	W =  90.000 deg,	P =   0.000 deg,	R =   90.000 deg
};
P[1718]{
   GP1:
	UF : 0, UT : 6,		CONFIG : 'N U T, 0, 0, 0',
	X =  65.499  mm,	Y =   -283.961  mm,	Z =   -229.185  mm,
	W =  90.000 deg,	P =   0.000 deg,	R =   90.000 deg
};
P[1719]{
   GP1:
	UF : 0, UT : 6,		CONFIG : 'N U T, 0, 0, 0',
	X =  64.374  mm,	Y =   -284.663  mm,	Z =   -229.314  mm,
	W =  90.000 deg,	P =   0.000 deg,	R =   90.000 deg
};
P[1720]{
   GP1:
	UF : 0, UT : 6,		CONFIG : 'N U T, 0, 0, 0',
	X =  62.334  mm,	Y =   -285.736  mm,	Z =   -229.059  mm,
	W =  90.000 deg,	P =   0.000 deg,	R =   90.000 deg
};
P[1721]{
   GP1:
	UF : 0, UT : 6,		CONFIG : 'N U T, 0, 0, 0',
	X =  61.528  mm,	Y =   -286.336  mm,	Z =   -229.385  mm,
	W =  90.000 deg,	P =   0.000 deg,	R =   90.000 deg
};
P[1722]{
   GP1:
	UF : 0, UT : 6,		CONFIG : 'N U T, 0, 0, 0',
	X =  60.500  mm,	Y =   -286.765  mm,	Z =   -228.984  mm,
	W =  90.000 deg,	P =   0.000 deg,	R =   90.000 deg
};
P[1723]{
   GP1:
	UF : 0, UT : 6,		CONFIG : 'N U T, 0, 0, 0',
	X =  59.972  mm,	Y =   -287.179  mm,	Z =   -229.250  mm,
	W =  90.000 deg,	P =   0.000 deg,	R =   90.000 deg
};
P[1724]{
   GP1:
	UF : 0, UT : 6,		CONFIG : 'N U T, 0, 0, 0',
	X =  58.339  mm,	Y =   -288.171  mm,	Z =   -229.370  mm,
	W =  90.000 deg,	P =   0.000 deg,	R =   90.000 deg
};
P[1725]{
   GP1:
	UF : 0, UT : 6,		CONFIG : 'N U T, 0, 0, 0',
	X =  53.179  mm,	Y =   -291.104  mm,	Z =   -229.258  mm,
	W =  90.000 deg,	P =   0.000 deg,	R =   90.000 deg
};
P[1726]{
   GP1:
	UF : 0, UT : 6,		CONFIG : 'N U T, 0, 0, 0',
	X =  52.446  mm,	Y =   -291.487  mm,	Z =   -229.159  mm,
	W =  90.000 deg,	P =   0.000 deg,	R =   90.000 deg
};
P[1727]{
   GP1:
	UF : 0, UT : 6,		CONFIG : 'N U T, 0, 0, 0',
	X =  50.068  mm,	Y =   -292.765  mm,	Z =   -228.929  mm,
	W =  90.000 deg,	P =   0.000 deg,	R =   90.000 deg
};
P[1728]{
   GP1:
	UF : 0, UT : 6,		CONFIG : 'N U T, 0, 0, 0',
	X =  47.155  mm,	Y =   -294.447  mm,	Z =   -228.929  mm,
	W =  90.000 deg,	P =   0.000 deg,	R =   90.000 deg
};
P[1729]{
   GP1:
	UF : 0, UT : 6,		CONFIG : 'N U T, 0, 0, 0',
	X =  45.389  mm,	Y =   -295.537  mm,	Z =   -229.099  mm,
	W =  90.000 deg,	P =   0.000 deg,	R =   90.000 deg
};
P[1730]{
   GP1:
	UF : 0, UT : 6,		CONFIG : 'N U T, 0, 0, 0',
	X =  41.975  mm,	Y =   -297.626  mm,	Z =   -229.386  mm,
	W =  90.000 deg,	P =   0.000 deg,	R =   90.000 deg
};
P[1731]{
   GP1:
	UF : 0, UT : 6,		CONFIG : 'N U T, 0, 0, 0',
	X =  40.743  mm,	Y =   -298.267  mm,	Z =   -229.217  mm,
	W =  90.000 deg,	P =   0.000 deg,	R =   90.000 deg
};
P[1732]{
   GP1:
	UF : 0, UT : 6,		CONFIG : 'N U T, 0, 0, 0',
	X =  39.529  mm,	Y =   -298.978  mm,	Z =   -229.239  mm,
	W =  90.000 deg,	P =   0.000 deg,	R =   90.000 deg
};
P[1733]{
   GP1:
	UF : 0, UT : 6,		CONFIG : 'N U T, 0, 0, 0',
	X =  38.765  mm,	Y =   -299.424  mm,	Z =   -229.251  mm,
	W =  90.000 deg,	P =   0.000 deg,	R =   90.000 deg
};
P[1734]{
   GP1:
	UF : 0, UT : 6,		CONFIG : 'N U T, 0, 0, 0',
	X =  37.888  mm,	Y =   -299.974  mm,	Z =   -229.356  mm,
	W =  90.000 deg,	P =   0.000 deg,	R =   90.000 deg
};
P[1735]{
   GP1:
	UF : 0, UT : 6,		CONFIG : 'N U T, 0, 0, 0',
	X =  37.310  mm,	Y =   -300.268  mm,	Z =   -229.259  mm,
	W =  90.000 deg,	P =   0.000 deg,	R =   90.000 deg
};
P[1736]{
   GP1:
	UF : 0, UT : 6,		CONFIG : 'N U T, 0, 0, 0',
	X =  36.423  mm,	Y =   -300.815  mm,	Z =   -229.344  mm,
	W =  90.000 deg,	P =   0.000 deg,	R =   90.000 deg
};
P[1737]{
   GP1:
	UF : 0, UT : 6,		CONFIG : 'N U T, 0, 0, 0',
	X =  34.210  mm,	Y =   -301.938  mm,	Z =   -228.969  mm,
	W =  90.000 deg,	P =   0.000 deg,	R =   90.000 deg
};
P[1738]{
   GP1:
	UF : 0, UT : 6,		CONFIG : 'N U T, 0, 0, 0',
	X =  31.437  mm,	Y =   -303.526  mm,	Z =   -228.939  mm,
	W =  90.000 deg,	P =   0.000 deg,	R =   90.000 deg
};
P[1739]{
   GP1:
	UF : 0, UT : 6,		CONFIG : 'N U T, 0, 0, 0',
	X =  30.762  mm,	Y =   -303.936  mm,	Z =   -228.988  mm,
	W =  90.000 deg,	P =   0.000 deg,	R =   90.000 deg
};
P[1740]{
   GP1:
	UF : 0, UT : 6,		CONFIG : 'N U T, 0, 0, 0',
	X =  30.126  mm,	Y =   -304.358  mm,	Z =   -229.121  mm,
	W =  90.000 deg,	P =   0.000 deg,	R =   90.000 deg
};
P[1741]{
   GP1:
	UF : 0, UT : 6,		CONFIG : 'N U T, 0, 0, 0',
	X =  29.321  mm,	Y =   -304.858  mm,	Z =   -229.206  mm,
	W =  90.000 deg,	P =   0.000 deg,	R =   90.000 deg
};
P[1742]{
   GP1:
	UF : 0, UT : 6,		CONFIG : 'N U T, 0, 0, 0',
	X =  28.546  mm,	Y =   -305.311  mm,	Z =   -229.219  mm,
	W =  90.000 deg,	P =   0.000 deg,	R =   90.000 deg
};
P[1743]{
   GP1:
	UF : 0, UT : 6,		CONFIG : 'N U T, 0, 0, 0',
	X =  26.880  mm,	Y =   -306.323  mm,	Z =   -229.338  mm,
	W =  90.000 deg,	P =   0.000 deg,	R =   90.000 deg
};
P[1744]{
   GP1:
	UF : 0, UT : 6,		CONFIG : 'N U T, 0, 0, 0',
	X =  24.918  mm,	Y =   -307.459  mm,	Z =   -229.349  mm,
	W =  90.000 deg,	P =   0.000 deg,	R =   90.000 deg
};
P[1745]{
   GP1:
	UF : 0, UT : 6,		CONFIG : 'N U T, 0, 0, 0',
	X =  24.359  mm,	Y =   -307.779  mm,	Z =   -229.343  mm,
	W =  90.000 deg,	P =   0.000 deg,	R =   90.000 deg
};
P[1746]{
   GP1:
	UF : 0, UT : 6,		CONFIG : 'N U T, 0, 0, 0',
	X =  23.494  mm,	Y =   -308.206  mm,	Z =   -229.165  mm,
	W =  90.000 deg,	P =   0.000 deg,	R =   90.000 deg
};
P[1747]{
   GP1:
	UF : 0, UT : 6,		CONFIG : 'N U T, 0, 0, 0',
	X =  22.302  mm,	Y =   -308.926  mm,	Z =   -229.240  mm,
	W =  90.000 deg,	P =   0.000 deg,	R =   90.000 deg
};
P[1748]{
   GP1:
	UF : 0, UT : 6,		CONFIG : 'N U T, 0, 0, 0',
	X =  20.679  mm,	Y =   -309.863  mm,	Z =   -229.241  mm,
	W =  90.000 deg,	P =   0.000 deg,	R =   90.000 deg
};
P[1749]{
   GP1:
	UF : 0, UT : 6,		CONFIG : 'N U T, 0, 0, 0',
	X =  17.947  mm,	Y =   -311.366  mm,	Z =   -229.061  mm,
	W =  90.000 deg,	P =   0.000 deg,	R =   90.000 deg
};
P[1750]{
   GP1:
	UF : 0, UT : 6,		CONFIG : 'N U T, 0, 0, 0',
	X =  15.569  mm,	Y =   -312.760  mm,	Z =   -229.113  mm,
	W =  90.000 deg,	P =   0.000 deg,	R =   90.000 deg
};
P[1751]{
   GP1:
	UF : 0, UT : 6,		CONFIG : 'N U T, 0, 0, 0',
	X =  12.896  mm,	Y =   -314.404  mm,	Z =   -229.357  mm,
	W =  90.000 deg,	P =   0.000 deg,	R =   90.000 deg
};
P[1752]{
   GP1:
	UF : 0, UT : 6,		CONFIG : 'N U T, 0, 0, 0',
	X =  11.173  mm,	Y =   -315.284  mm,	Z =   -229.077  mm,
	W =  90.000 deg,	P =   0.000 deg,	R =   90.000 deg
};
P[1753]{
   GP1:
	UF : 0, UT : 6,		CONFIG : 'N U T, 0, 0, 0',
	X =  9.686  mm,	Y =   -316.168  mm,	Z =   -229.140  mm,
	W =  90.000 deg,	P =   0.000 deg,	R =   90.000 deg
};
P[1754]{
   GP1:
	UF : 0, UT : 6,		CONFIG : 'N U T, 0, 0, 0',
	X =  8.873  mm,	Y =   -316.625  mm,	Z =   -229.112  mm,
	W =  90.000 deg,	P =   0.000 deg,	R =   90.000 deg
};
P[1755]{
   GP1:
	UF : 0, UT : 6,		CONFIG : 'N U T, 0, 0, 0',
	X =  8.041  mm,	Y =   -317.205  mm,	Z =   -229.351  mm,
	W =  90.000 deg,	P =   0.000 deg,	R =   90.000 deg
};
P[1756]{
   GP1:
	UF : 0, UT : 6,		CONFIG : 'N U T, 0, 0, 0',
	X =  6.642  mm,	Y =   -317.970  mm,	Z =   -229.246  mm,
	W =  90.000 deg,	P =   0.000 deg,	R =   90.000 deg
};
P[1757]{
   GP1:
	UF : 0, UT : 6,		CONFIG : 'N U T, 0, 0, 0',
	X =  5.653  mm,	Y =   -318.591  mm,	Z =   -229.370  mm,
	W =  90.000 deg,	P =   0.000 deg,	R =   90.000 deg
};
P[1758]{
   GP1:
	UF : 0, UT : 6,		CONFIG : 'N U T, 0, 0, 0',
	X =  4.796  mm,	Y =   -318.944  mm,	Z =   -229.023  mm,
	W =  90.000 deg,	P =   0.000 deg,	R =   90.000 deg
};
P[1759]{
   GP1:
	UF : 0, UT : 6,		CONFIG : 'N U T, 0, 0, 0',
	X =  3.388  mm,	Y =   -319.857  mm,	Z =   -229.269  mm,
	W =  90.000 deg,	P =   0.000 deg,	R =   90.000 deg
};
P[1760]{
   GP1:
	UF : 0, UT : 6,		CONFIG : 'N U T, 0, 0, 0',
	X =  2.077  mm,	Y =   -320.526  mm,	Z =   -229.055  mm,
	W =  90.000 deg,	P =   0.000 deg,	R =   90.000 deg
};
P[1761]{
   GP1:
	UF : 0, UT : 6,		CONFIG : 'N U T, 0, 0, 0',
	X =  0.657  mm,	Y =   -321.382  mm,	Z =   -229.142  mm,
	W =  90.000 deg,	P =   0.000 deg,	R =   90.000 deg
};
P[1762]{
   GP1:
	UF : 0, UT : 6,		CONFIG : 'N U T, 0, 0, 0',
	X =  -0.741  mm,	Y =   -322.160  mm,	Z =   -229.070  mm,
	W =  90.000 deg,	P =   0.000 deg,	R =   90.000 deg
};
P[1763]{
   GP1:
	UF : 0, UT : 6,		CONFIG : 'N U T, 0, 0, 0',
	X =  -1.523  mm,	Y =   -322.657  mm,	Z =   -229.181  mm,
	W =  90.000 deg,	P =   0.000 deg,	R =   90.000 deg
};
P[1764]{
   GP1:
	UF : 0, UT : 6,		CONFIG : 'N U T, 0, 0, 0',
	X =  -2.343  mm,	Y =   -323.167  mm,	Z =   -229.270  mm,
	W =  90.000 deg,	P =   0.000 deg,	R =   90.000 deg
};
P[1765]{
   GP1:
	UF : 0, UT : 6,		CONFIG : 'N U T, 0, 0, 0',
	X =  -3.964  mm,	Y =   -323.984  mm,	Z =   -228.981  mm,
	W =  90.000 deg,	P =   0.000 deg,	R =   90.000 deg
};
P[1766]{
   GP1:
	UF : 0, UT : 6,		CONFIG : 'N U T, 0, 0, 0',
	X =  -6.538  mm,	Y =   -325.534  mm,	Z =   -229.136  mm,
	W =  90.000 deg,	P =   0.000 deg,	R =   90.000 deg
};
P[1767]{
   GP1:
	UF : 0, UT : 6,		CONFIG : 'N U T, 0, 0, 0',
	X =  -7.592  mm,	Y =   -326.225  mm,	Z =   -229.338  mm,
	W =  90.000 deg,	P =   0.000 deg,	R =   90.000 deg
};
P[1768]{
   GP1:
	UF : 0, UT : 6,		CONFIG : 'N U T, 0, 0, 0',
	X =  -12.691  mm,	Y =   -329.122  mm,	Z =   -229.220  mm,
	W =  90.000 deg,	P =   0.000 deg,	R =   90.000 deg
};
P[1769]{
   GP1:
	UF : 0, UT : 6,		CONFIG : 'N U T, 0, 0, 0',
	X =  -13.895  mm,	Y =   -329.816  mm,	Z =   -229.218  mm,
	W =  90.000 deg,	P =   0.000 deg,	R =   90.000 deg
};
P[1770]{
   GP1:
	UF : 0, UT : 6,		CONFIG : 'N U T, 0, 0, 0',
	X =  -14.816  mm,	Y =   -330.402  mm,	Z =   -229.349  mm,
	W =  90.000 deg,	P =   0.000 deg,	R =   90.000 deg
};
P[1771]{
   GP1:
	UF : 0, UT : 6,		CONFIG : 'N U T, 0, 0, 0',
	X =  -15.958  mm,	Y =   -330.974  mm,	Z =   -229.139  mm,
	W =  90.000 deg,	P =   0.000 deg,	R =   90.000 deg
};
P[1772]{
   GP1:
	UF : 0, UT : 6,		CONFIG : 'N U T, 0, 0, 0',
	X =  -17.640  mm,	Y =   -331.967  mm,	Z =   -229.191  mm,
	W =  90.000 deg,	P =   0.000 deg,	R =   90.000 deg
};
P[1773]{
   GP1:
	UF : 0, UT : 6,		CONFIG : 'N U T, 0, 0, 0',
	X =  -19.082  mm,	Y =   -332.836  mm,	Z =   -229.281  mm,
	W =  90.000 deg,	P =   0.000 deg,	R =   90.000 deg
};
P[1774]{
   GP1:
	UF : 0, UT : 6,		CONFIG : 'N U T, 0, 0, 0',
	X =  -19.863  mm,	Y =   -333.279  mm,	Z =   -229.261  mm,
	W =  90.000 deg,	P =   0.000 deg,	R =   90.000 deg
};
P[1775]{
   GP1:
	UF : 0, UT : 6,		CONFIG : 'N U T, 0, 0, 0',
	X =  -21.186  mm,	Y =   -333.972  mm,	Z =   -229.088  mm,
	W =  90.000 deg,	P =   0.000 deg,	R =   90.000 deg
};
P[1776]{
   GP1:
	UF : 0, UT : 6,		CONFIG : 'N U T, 0, 0, 0',
	X =  -22.635  mm,	Y =   -334.894  mm,	Z =   -229.296  mm,
	W =  90.000 deg,	P =   0.000 deg,	R =   90.000 deg
};
P[1777]{
   GP1:
	UF : 0, UT : 6,		CONFIG : 'N U T, 0, 0, 0',
	X =  -24.157  mm,	Y =   -335.703  mm,	Z =   -229.127  mm,
	W =  90.000 deg,	P =   0.000 deg,	R =   90.000 deg
};
P[1778]{
   GP1:
	UF : 0, UT : 6,		CONFIG : 'N U T, 0, 0, 0',
	X =  -25.039  mm,	Y =   -336.224  mm,	Z =   -229.155  mm,
	W =  90.000 deg,	P =   0.000 deg,	R =   90.000 deg
};
P[1779]{
   GP1:
	UF : 0, UT : 6,		CONFIG : 'N U T, 0, 0, 0',
	X =  -25.704  mm,	Y =   -336.510  mm,	Z =   -228.916  mm,
	W =  90.000 deg,	P =   0.000 deg,	R =   90.000 deg
};
P[1780]{
   GP1:
	UF : 0, UT : 6,		CONFIG : 'N U T, 0, 0, 0',
	X =  -26.496  mm,	Y =   -337.068  mm,	Z =   -229.160  mm,
	W =  90.000 deg,	P =   0.000 deg,	R =   90.000 deg
};
P[1781]{
   GP1:
	UF : 0, UT : 6,		CONFIG : 'N U T, 0, 0, 0',
	X =  -29.082  mm,	Y =   -338.564  mm,	Z =   -229.168  mm,
	W =  90.000 deg,	P =   0.000 deg,	R =   90.000 deg
};
P[1782]{
   GP1:
	UF : 0, UT : 6,		CONFIG : 'N U T, 0, 0, 0',
	X =  -32.694  mm,	Y =   -340.689  mm,	Z =   -229.266  mm,
	W =  90.000 deg,	P =   0.000 deg,	R =   90.000 deg
};
P[1783]{
   GP1:
	UF : 0, UT : 6,		CONFIG : 'N U T, 0, 0, 0',
	X =  -33.349  mm,	Y =   -341.119  mm,	Z =   -229.387  mm,
	W =  90.000 deg,	P =   0.000 deg,	R =   90.000 deg
};
P[1784]{
   GP1:
	UF : 0, UT : 6,		CONFIG : 'N U T, 0, 0, 0',
	X =  -38.216  mm,	Y =   -343.745  mm,	Z =   -228.944  mm,
	W =  90.000 deg,	P =   0.000 deg,	R =   90.000 deg
};
P[1785]{
   GP1:
	UF : 0, UT : 6,		CONFIG : 'N U T, 0, 0, 0',
	X =  -41.561  mm,	Y =   -345.684  mm,	Z =   -228.963  mm,
	W =  90.000 deg,	P =   0.000 deg,	R =   90.000 deg
};
P[1786]{
   GP1:
	UF : 0, UT : 6,		CONFIG : 'N U T, 0, 0, 0',
	X =  -42.055  mm,	Y =   -346.140  mm,	Z =   -229.376  mm,
	W =  90.000 deg,	P =   0.000 deg,	R =   90.000 deg
};
P[1787]{
   GP1:
	UF : 0, UT : 6,		CONFIG : 'N U T, 0, 0, 0',
	X =  -42.732  mm,	Y =   -346.389  mm,	Z =   -229.030  mm,
	W =  90.000 deg,	P =   0.000 deg,	R =   90.000 deg
};
P[1788]{
   GP1:
	UF : 0, UT : 6,		CONFIG : 'N U T, 0, 0, 0',
	X =  -43.777  mm,	Y =   -347.079  mm,	Z =   -229.241  mm,
	W =  90.000 deg,	P =   0.000 deg,	R =   90.000 deg
};
P[1789]{
   GP1:
	UF : 0, UT : 6,		CONFIG : 'N U T, 0, 0, 0',
	X =  -44.518  mm,	Y =   -347.535  mm,	Z =   -229.311  mm,
	W =  90.000 deg,	P =   0.000 deg,	R =   90.000 deg
};
P[1790]{
   GP1:
	UF : 0, UT : 6,		CONFIG : 'N U T, 0, 0, 0',
	X =  -45.258  mm,	Y =   -347.966  mm,	Z =   -229.318  mm,
	W =  90.000 deg,	P =   0.000 deg,	R =   90.000 deg
};
P[1791]{
   GP1:
	UF : 0, UT : 6,		CONFIG : 'N U T, 0, 0, 0',
	X =  -46.748  mm,	Y =   -348.709  mm,	Z =   -229.034  mm,
	W =  90.000 deg,	P =   0.000 deg,	R =   90.000 deg
};
P[1792]{
   GP1:
	UF : 0, UT : 6,		CONFIG : 'N U T, 0, 0, 0',
	X =  -50.185  mm,	Y =   -350.794  mm,	Z =   -229.276  mm,
	W =  90.000 deg,	P =   0.000 deg,	R =   90.000 deg
};
P[1793]{
   GP1:
	UF : 0, UT : 6,		CONFIG : 'N U T, 0, 0, 0',
	X =  -50.896  mm,	Y =   -351.228  mm,	Z =   -229.333  mm,
	W =  90.000 deg,	P =   0.000 deg,	R =   90.000 deg
};
P[1794]{
   GP1:
	UF : 0, UT : 6,		CONFIG : 'N U T, 0, 0, 0',
	X =  -51.979  mm,	Y =   -351.709  mm,	Z =   -228.984  mm,
	W =  90.000 deg,	P =   0.000 deg,	R =   90.000 deg
};
P[1795]{
   GP1:
	UF : 0, UT : 6,		CONFIG : 'N U T, 0, 0, 0',
	X =  -54.128  mm,	Y =   -353.013  mm,	Z =   -229.137  mm,
	W =  90.000 deg,	P =   0.000 deg,	R =   90.000 deg
};
P[1796]{
   GP1:
	UF : 0, UT : 6,		CONFIG : 'N U T, 0, 0, 0',
	X =  -54.799  mm,	Y =   -353.441  mm,	Z =   -229.237  mm,
	W =  90.000 deg,	P =   0.000 deg,	R =   90.000 deg
};
P[1797]{
   GP1:
	UF : 0, UT : 6,		CONFIG : 'N U T, 0, 0, 0',
	X =  -55.346  mm,	Y =   -353.813  mm,	Z =   -229.371  mm,
	W =  90.000 deg,	P =   0.000 deg,	R =   90.000 deg
};
P[1798]{
   GP1:
	UF : 0, UT : 6,		CONFIG : 'N U T, 0, 0, 0',
	X =  -59.610  mm,	Y =   -356.160  mm,	Z =   -229.092  mm,
	W =  90.000 deg,	P =   0.000 deg,	R =   90.000 deg
};
P[1799]{
   GP1:
	UF : 0, UT : 6,		CONFIG : 'N U T, 0, 0, 0',
	X =  -60.201  mm,	Y =   -356.446  mm,	Z =   -228.959  mm,
	W =  90.000 deg,	P =   0.000 deg,	R =   90.000 deg
};
P[1800]{
   GP1:
	UF : 0, UT : 6,		CONFIG : 'N U T, 0, 0, 0',
	X =  -61.122  mm,	Y =   -357.104  mm,	Z =   -229.266  mm,
	W =  90.000 deg,	P =   0.000 deg,	R =   90.000 deg
};
P[1801]{
   GP1:
	UF : 0, UT : 6,		CONFIG : 'N U T, 0, 0, 0',
	X =  -62.393  mm,	Y =   -357.747  mm,	Z =   -229.045  mm,
	W =  90.000 deg,	P =   0.000 deg,	R =   90.000 deg
};
P[1802]{
   GP1:
	UF : 0, UT : 6,		CONFIG : 'N U T, 0, 0, 0',
	X =  -63.618  mm,	Y =   -358.533  mm,	Z =   -229.238  mm,
	W =  90.000 deg,	P =   0.000 deg,	R =   90.000 deg
};
P[1803]{
   GP1:
	UF : 0, UT : 6,		CONFIG : 'N U T, 0, 0, 0',
	X =  -64.685  mm,	Y =   -359.172  mm,	Z =   -229.293  mm,
	W =  90.000 deg,	P =   0.000 deg,	R =   90.000 deg
};
P[1804]{
   GP1:
	UF : 0, UT : 6,		CONFIG : 'N U T, 0, 0, 0',
	X =  -65.434  mm,	Y =   -359.590  mm,	Z =   -229.257  mm,
	W =  90.000 deg,	P =   0.000 deg,	R =   90.000 deg
};
P[1805]{
   GP1:
	UF : 0, UT : 6,		CONFIG : 'N U T, 0, 0, 0',
	X =  -67.552  mm,	Y =   -360.821  mm,	Z =   -229.277  mm,
	W =  90.000 deg,	P =   0.000 deg,	R =   90.000 deg
};
P[1806]{
   GP1:
	UF : 0, UT : 6,		CONFIG : 'N U T, 0, 0, 0',
	X =  -68.252  mm,	Y =   -361.161  mm,	Z =   -229.121  mm,
	W =  90.000 deg,	P =   0.000 deg,	R =   90.000 deg
};
P[1807]{
   GP1:
	UF : 0, UT : 6,		CONFIG : 'N U T, 0, 0, 0',
	X =  -69.737  mm,	Y =   -361.996  mm,	Z =   -229.066  mm,
	W =  90.000 deg,	P =   0.000 deg,	R =   90.000 deg
};
P[1808]{
   GP1:
	UF : 0, UT : 6,		CONFIG : 'N U T, 0, 0, 0',
	X =  -71.695  mm,	Y =   -363.184  mm,	Z =   -229.206  mm,
	W =  90.000 deg,	P =   0.000 deg,	R =   90.000 deg
};
P[1809]{
   GP1:
	UF : 0, UT : 6,		CONFIG : 'N U T, 0, 0, 0',
	X =  -73.384  mm,	Y =   -364.195  mm,	Z =   -229.294  mm,
	W =  90.000 deg,	P =   0.000 deg,	R =   90.000 deg
};
P[1810]{
   GP1:
	UF : 0, UT : 6,		CONFIG : 'N U T, 0, 0, 0',
	X =  -74.673  mm,	Y =   -364.878  mm,	Z =   -229.144  mm,
	W =  90.000 deg,	P =   0.000 deg,	R =   90.000 deg
};
P[1811]{
   GP1:
	UF : 0, UT : 6,		CONFIG : 'N U T, 0, 0, 0',
	X =  -76.471  mm,	Y =   -365.928  mm,	Z =   -229.173  mm,
	W =  90.000 deg,	P =   0.000 deg,	R =   90.000 deg
};
P[1812]{
   GP1:
	UF : 0, UT : 6,		CONFIG : 'N U T, 0, 0, 0',
	X =  -78.015  mm,	Y =   -366.782  mm,	Z =   -229.082  mm,
	W =  90.000 deg,	P =   0.000 deg,	R =   90.000 deg
};
P[1813]{
   GP1:
	UF : 0, UT : 6,		CONFIG : 'N U T, 0, 0, 0',
	X =  -82.837  mm,	Y =   -369.534  mm,	Z =   -229.004  mm,
	W =  90.000 deg,	P =   0.000 deg,	R =   90.000 deg
};
P[1814]{
   GP1:
	UF : 0, UT : 6,		CONFIG : 'N U T, 0, 0, 0',
	X =  -83.583  mm,	Y =   -369.935  mm,	Z =   -228.932  mm,
	W =  90.000 deg,	P =   0.000 deg,	R =   90.000 deg
};
P[1815]{
   GP1:
	UF : 0, UT : 6,		CONFIG : 'N U T, 0, 0, 0',
	X =  -85.190  mm,	Y =   -370.941  mm,	Z =   -229.121  mm,
	W =  90.000 deg,	P =   0.000 deg,	R =   90.000 deg
};
P[1816]{
   GP1:
	UF : 0, UT : 6,		CONFIG : 'N U T, 0, 0, 0',
	X =  -86.946  mm,	Y =   -371.886  mm,	Z =   -228.955  mm,
	W =  90.000 deg,	P =   0.000 deg,	R =   90.000 deg
};
P[1817]{
   GP1:
	UF : 0, UT : 6,		CONFIG : 'N U T, 0, 0, 0',
	X =  -87.736  mm,	Y =   -372.509  mm,	Z =   -229.360  mm,
	W =  90.000 deg,	P =   0.000 deg,	R =   90.000 deg
};
P[1818]{
   GP1:
	UF : 0, UT : 6,		CONFIG : 'N U T, 0, 0, 0',
	X =  -89.887  mm,	Y =   -373.748  mm,	Z =   -229.351  mm,
	W =  90.000 deg,	P =   0.000 deg,	R =   90.000 deg
};
P[1819]{
   GP1:
	UF : 0, UT : 6,		CONFIG : 'N U T, 0, 0, 0',
	X =  -91.030  mm,	Y =   -374.267  mm,	Z =   -229.010  mm,
	W =  90.000 deg,	P =   0.000 deg,	R =   90.000 deg
};
P[1820]{
   GP1:
	UF : 0, UT : 6,		CONFIG : 'N U T, 0, 0, 0',
	X =  -94.361  mm,	Y =   -376.300  mm,	Z =   -229.274  mm,
	W =  90.000 deg,	P =   0.000 deg,	R =   90.000 deg
};
P[1821]{
   GP1:
	UF : 0, UT : 6,		CONFIG : 'N U T, 0, 0, 0',
	X =  -96.414  mm,	Y =   -377.422  mm,	Z =   -229.121  mm,
	W =  90.000 deg,	P =   0.000 deg,	R =   90.000 deg
};
P[1822]{
   GP1:
	UF : 0, UT : 6,		CONFIG : 'N U T, 0, 0, 0',
	X =  -98.002  mm,	Y =   -378.340  mm,	Z =   -229.123  mm,
	W =  90.000 deg,	P =   0.000 deg,	R =   90.000 deg
};
P[1823]{
   GP1:
	UF : 0, UT : 6,		CONFIG : 'N U T, 0, 0, 0',
	X =  -101.725  mm,	Y =   -380.543  mm,	Z =   -229.255  mm,
	W =  90.000 deg,	P =   0.000 deg,	R =   90.000 deg
};
P[1824]{
   GP1:
	UF : 0, UT : 6,		CONFIG : 'N U T, 0, 0, 0',
	X =  -102.580  mm,	Y =   -381.019  mm,	Z =   -229.211  mm,
	W =  90.000 deg,	P =   0.000 deg,	R =   90.000 deg
};
P[1825]{
   GP1:
	UF : 0, UT : 6,		CONFIG : 'N U T, 0, 0, 0',
	X =  -103.214  mm,	Y =   -381.274  mm,	Z =   -228.942  mm,
	W =  90.000 deg,	P =   0.000 deg,	R =   90.000 deg
};
P[1826]{
   GP1:
	UF : 0, UT : 6,		CONFIG : 'N U T, 0, 0, 0',
	X =  -104.057  mm,	Y =   -381.765  mm,	Z =   -228.951  mm,
	W =  90.000 deg,	P =   0.000 deg,	R =   90.000 deg
};
P[1827]{
   GP1:
	UF : 0, UT : 6,		CONFIG : 'N U T, 0, 0, 0',
	X =  -104.771  mm,	Y =   -382.207  mm,	Z =   -229.023  mm,
	W =  90.000 deg,	P =   0.000 deg,	R =   90.000 deg
};
P[1828]{
   GP1:
	UF : 0, UT : 6,		CONFIG : 'N U T, 0, 0, 0',
	X =  -106.220  mm,	Y =   -383.159  mm,	Z =   -229.305  mm,
	W =  90.000 deg,	P =   0.000 deg,	R =   90.000 deg
};
P[1829]{
   GP1:
	UF : 0, UT : 6,		CONFIG : 'N U T, 0, 0, 0',
	X =  -107.258  mm,	Y =   -383.655  mm,	Z =   -229.053  mm,
	W =  90.000 deg,	P =   0.000 deg,	R =   90.000 deg
};
P[1830]{
   GP1:
	UF : 0, UT : 6,		CONFIG : 'N U T, 0, 0, 0',
	X =  -108.626  mm,	Y =   -384.389  mm,	Z =   -228.918  mm,
	W =  90.000 deg,	P =   0.000 deg,	R =   90.000 deg
};
P[1831]{
   GP1:
	UF : 0, UT : 6,		CONFIG : 'N U T, 0, 0, 0',
	X =  -110.424  mm,	Y =   -385.480  mm,	Z =   -229.046  mm,
	W =  90.000 deg,	P =   0.000 deg,	R =   90.000 deg
};
P[1832]{
   GP1:
	UF : 0, UT : 6,		CONFIG : 'N U T, 0, 0, 0',
	X =  -111.106  mm,	Y =   -385.858  mm,	Z =   -228.907  mm,
	W =  90.000 deg,	P =   0.000 deg,	R =   90.000 deg
};
P[1833]{
   GP1:
	UF : 0, UT : 6,		CONFIG : 'N U T, 0, 0, 0',
	X =  -111.846  mm,	Y =   -386.429  mm,	Z =   -229.006  mm,
	W =  90.000 deg,	P =   0.000 deg,	R =   90.000 deg
};
P[1834]{
   GP1:
	UF : 0, UT : 6,		CONFIG : 'N U T, 0, 0, 0',
	X =  -114.050  mm,	Y =   -388.372  mm,	Z =   -229.002  mm,
	W =  90.000 deg,	P =   0.000 deg,	R =   90.000 deg
};
P[1835]{
   GP1:
	UF : 0, UT : 6,		CONFIG : 'N U T, 0, 0, 0',
	X =  -115.101  mm,	Y =   -389.696  mm,	Z =   -228.999  mm,
	W =  90.000 deg,	P =   0.000 deg,	R =   90.000 deg
};
P[1836]{
   GP1:
	UF : 0, UT : 6,		CONFIG : 'N U T, 0, 0, 0',
	X =  -115.762  mm,	Y =   -390.707  mm,	Z =   -228.966  mm,
	W =  90.000 deg,	P =   0.000 deg,	R =   90.000 deg
};
P[1837]{
   GP1:
	UF : 0, UT : 6,		CONFIG : 'N U T, 0, 0, 0',
	X =  -116.815  mm,	Y =   -393.661  mm,	Z =   -229.189  mm,
	W =  90.000 deg,	P =   0.000 deg,	R =   90.000 deg
};
P[1838]{
   GP1:
	UF : 0, UT : 6,		CONFIG : 'N U T, 0, 0, 0',
	X =  -116.981  mm,	Y =   -394.369  mm,	Z =   -229.133  mm,
	W =  90.000 deg,	P =   0.000 deg,	R =   90.000 deg
};
P[1839]{
   GP1:
	UF : 0, UT : 6,		CONFIG : 'N U T, 0, 0, 0',
	X =  -117.216  mm,	Y =   -397.476  mm,	Z =   -229.036  mm,
	W =  90.000 deg,	P =   0.000 deg,	R =   90.000 deg
};
P[1840]{
   GP1:
	UF : 0, UT : 6,		CONFIG : 'N U T, 0, 0, 0',
	X =  -117.144  mm,	Y =   -398.247  mm,	Z =   -229.117  mm,
	W =  90.000 deg,	P =   0.000 deg,	R =   90.000 deg
};
P[1841]{
   GP1:
	UF : 0, UT : 6,		CONFIG : 'N U T, 0, 0, 0',
	X =  -116.699  mm,	Y =   -400.629  mm,	Z =   -228.902  mm,
	W =  90.000 deg,	P =   0.000 deg,	R =   90.000 deg
};
P[1842]{
   GP1:
	UF : 0, UT : 6,		CONFIG : 'N U T, 0, 0, 0',
	X =  -115.143  mm,	Y =   -403.741  mm,	Z =   -229.218  mm,
	W =  90.000 deg,	P =   0.000 deg,	R =   90.000 deg
};
P[1843]{
   GP1:
	UF : 0, UT : 6,		CONFIG : 'N U T, 0, 0, 0',
	X =  -114.830  mm,	Y =   -404.473  mm,	Z =   -228.955  mm,
	W =  90.000 deg,	P =   0.000 deg,	R =   90.000 deg
};
P[1844]{
   GP1:
	UF : 0, UT : 6,		CONFIG : 'N U T, 0, 0, 0',
	X =  -114.278  mm,	Y =   -405.145  mm,	Z =   -229.351  mm,
	W =  90.000 deg,	P =   0.000 deg,	R =   90.000 deg
};
P[1845]{
   GP1:
	UF : 0, UT : 6,		CONFIG : 'N U T, 0, 0, 0',
	X =  -113.583  mm,	Y =   -406.477  mm,	Z =   -229.173  mm,
	W =  90.000 deg,	P =   0.000 deg,	R =   90.000 deg
};
P[1846]{
   GP1:
	UF : 0, UT : 6,		CONFIG : 'N U T, 0, 0, 0',
	X =  -111.947  mm,	Y =   -409.195  mm,	Z =   -229.335  mm,
	W =  90.000 deg,	P =   0.000 deg,	R =   90.000 deg
};
P[1847]{
   GP1:
	UF : 0, UT : 6,		CONFIG : 'N U T, 0, 0, 0',
	X =  -110.907  mm,	Y =   -411.061  mm,	Z =   -229.245  mm,
	W =  90.000 deg,	P =   0.000 deg,	R =   90.000 deg
};
P[1848]{
   GP1:
	UF : 0, UT : 6,		CONFIG : 'N U T, 0, 0, 0',
	X =  -110.205  mm,	Y =   -412.176  mm,	Z =   -229.385  mm,
	W =  90.000 deg,	P =   0.000 deg,	R =   90.000 deg
};
P[1849]{
   GP1:
	UF : 0, UT : 6,		CONFIG : 'N U T, 0, 0, 0',
	X =  -109.969  mm,	Y =   -412.840  mm,	Z =   -229.026  mm,
	W =  90.000 deg,	P =   0.000 deg,	R =   90.000 deg
};
P[1850]{
   GP1:
	UF : 0, UT : 6,		CONFIG : 'N U T, 0, 0, 0',
	X =  -108.686  mm,	Y =   -415.006  mm,	Z =   -229.104  mm,
	W =  90.000 deg,	P =   0.000 deg,	R =   90.000 deg
};
P[1851]{
   GP1:
	UF : 0, UT : 6,		CONFIG : 'N U T, 0, 0, 0',
	X =  -108.139  mm,	Y =   -415.790  mm,	Z =   -229.334  mm,
	W =  90.000 deg,	P =   0.000 deg,	R =   90.000 deg
};
P[1852]{
   GP1:
	UF : 0, UT : 6,		CONFIG : 'N U T, 0, 0, 0',
	X =  -107.446  mm,	Y =   -417.150  mm,	Z =   -229.110  mm,
	W =  90.000 deg,	P =   0.000 deg,	R =   90.000 deg
};
P[1853]{
   GP1:
	UF : 0, UT : 6,		CONFIG : 'N U T, 0, 0, 0',
	X =  -106.777  mm,	Y =   -418.198  mm,	Z =   -229.266  mm,
	W =  90.000 deg,	P =   0.000 deg,	R =   90.000 deg
};
P[1854]{
   GP1:
	UF : 0, UT : 6,		CONFIG : 'N U T, 0, 0, 0',
	X =  -105.715  mm,	Y =   -419.969  mm,	Z =   -229.362  mm,
	W =  90.000 deg,	P =   0.000 deg,	R =   90.000 deg
};
P[1855]{
   GP1:
	UF : 0, UT : 6,		CONFIG : 'N U T, 0, 0, 0',
	X =  -102.894  mm,	Y =   -424.877  mm,	Z =   -229.333  mm,
	W =  90.000 deg,	P =   0.000 deg,	R =   90.000 deg
};
P[1856]{
   GP1:
	UF : 0, UT : 6,		CONFIG : 'N U T, 0, 0, 0',
	X =  -101.587  mm,	Y =   -427.111  mm,	Z =   -229.370  mm,
	W =  90.000 deg,	P =   0.000 deg,	R =   90.000 deg
};
P[1857]{
   GP1:
	UF : 0, UT : 6,		CONFIG : 'N U T, 0, 0, 0',
	X =  -101.111  mm,	Y =   -428.222  mm,	Z =   -228.971  mm,
	W =  90.000 deg,	P =   0.000 deg,	R =   90.000 deg
};
P[1858]{
   GP1:
	UF : 0, UT : 6,		CONFIG : 'N U T, 0, 0, 0',
	X =  -100.738  mm,	Y =   -428.828  mm,	Z =   -229.025  mm,
	W =  90.000 deg,	P =   0.000 deg,	R =   90.000 deg
};
P[1859]{
   GP1:
	UF : 0, UT : 6,		CONFIG : 'N U T, 0, 0, 0',
	X =  -100.382  mm,	Y =   -429.496  mm,	Z =   -228.954  mm,
	W =  90.000 deg,	P =   0.000 deg,	R =   90.000 deg
};
P[1860]{
   GP1:
	UF : 0, UT : 6,		CONFIG : 'N U T, 0, 0, 0',
	X =  -99.771  mm,	Y =   -430.443  mm,	Z =   -229.108  mm,
	W =  90.000 deg,	P =   0.000 deg,	R =   90.000 deg
};
P[1861]{
   GP1:
	UF : 0, UT : 6,		CONFIG : 'N U T, 0, 0, 0',
	X =  -97.945  mm,	Y =   -433.610  mm,	Z =   -229.104  mm,
	W =  90.000 deg,	P =   0.000 deg,	R =   90.000 deg
};
P[1862]{
   GP1:
	UF : 0, UT : 6,		CONFIG : 'N U T, 0, 0, 0',
	X =  -96.878  mm,	Y =   -435.314  mm,	Z =   -229.304  mm,
	W =  90.000 deg,	P =   0.000 deg,	R =   90.000 deg
};
P[1863]{
   GP1:
	UF : 0, UT : 6,		CONFIG : 'N U T, 0, 0, 0',
	X =  -95.918  mm,	Y =   -437.015  mm,	Z =   -229.252  mm,
	W =  90.000 deg,	P =   0.000 deg,	R =   90.000 deg
};
P[1864]{
   GP1:
	UF : 0, UT : 6,		CONFIG : 'N U T, 0, 0, 0',
	X =  -95.734  mm,	Y =   -437.573  mm,	Z =   -228.916  mm,
	W =  90.000 deg,	P =   0.000 deg,	R =   90.000 deg
};
P[1865]{
   GP1:
	UF : 0, UT : 6,		CONFIG : 'N U T, 0, 0, 0',
	X =  -94.251  mm,	Y =   -440.013  mm,	Z =   -229.096  mm,
	W =  90.000 deg,	P =   0.000 deg,	R =   90.000 deg
};
P[1866]{
   GP1:
	UF : 0, UT : 6,		CONFIG : 'N U T, 0, 0, 0',
	X =  -93.487  mm,	Y =   -441.177  mm,	Z =   -229.317  mm,
	W =  90.000 deg,	P =   0.000 deg,	R =   90.000 deg
};
P[1867]{
   GP1:
	UF : 0, UT : 6,		CONFIG : 'N U T, 0, 0, 0',
	X =  -92.630  mm,	Y =   -442.709  mm,	Z =   -229.251  mm,
	W =  90.000 deg,	P =   0.000 deg,	R =   90.000 deg
};
P[1868]{
   GP1:
	UF : 0, UT : 6,		CONFIG : 'N U T, 0, 0, 0',
	X =  -92.385  mm,	Y =   -443.308  mm,	Z =   -229.007  mm,
	W =  90.000 deg,	P =   0.000 deg,	R =   90.000 deg
};
P[1869]{
   GP1:
	UF : 0, UT : 6,		CONFIG : 'N U T, 0, 0, 0',
	X =  -91.614  mm,	Y =   -444.506  mm,	Z =   -229.201  mm,
	W =  90.000 deg,	P =   0.000 deg,	R =   90.000 deg
};
P[1870]{
   GP1:
	UF : 0, UT : 6,		CONFIG : 'N U T, 0, 0, 0',
	X =  -91.022  mm,	Y =   -445.447  mm,	Z =   -229.318  mm,
	W =  90.000 deg,	P =   0.000 deg,	R =   90.000 deg
};
P[1871]{
   GP1:
	UF : 0, UT : 6,		CONFIG : 'N U T, 0, 0, 0',
	X =  -90.796  mm,	Y =   -446.031  mm,	Z =   -229.048  mm,
	W =  90.000 deg,	P =   0.000 deg,	R =   90.000 deg
};
P[1872]{
   GP1:
	UF : 0, UT : 6,		CONFIG : 'N U T, 0, 0, 0',
	X =  -89.661  mm,	Y =   -447.816  mm,	Z =   -229.302  mm,
	W =  90.000 deg,	P =   0.000 deg,	R =   90.000 deg
};
P[1873]{
   GP1:
	UF : 0, UT : 6,		CONFIG : 'N U T, 0, 0, 0',
	X =  -88.469  mm,	Y =   -450.093  mm,	Z =   -229.002  mm,
	W =  90.000 deg,	P =   0.000 deg,	R =   90.000 deg
};
P[1874]{
   GP1:
	UF : 0, UT : 6,		CONFIG : 'N U T, 0, 0, 0',
	X =  -87.738  mm,	Y =   -451.149  mm,	Z =   -229.299  mm,
	W =  90.000 deg,	P =   0.000 deg,	R =   90.000 deg
};
P[1875]{
   GP1:
	UF : 0, UT : 6,		CONFIG : 'N U T, 0, 0, 0',
	X =  -86.732  mm,	Y =   -452.944  mm,	Z =   -229.224  mm,
	W =  90.000 deg,	P =   0.000 deg,	R =   90.000 deg
};
P[1876]{
   GP1:
	UF : 0, UT : 6,		CONFIG : 'N U T, 0, 0, 0',
	X =  -85.455  mm,	Y =   -455.178  mm,	Z =   -229.193  mm,
	W =  90.000 deg,	P =   0.000 deg,	R =   90.000 deg
};
P[1877]{
   GP1:
	UF : 0, UT : 6,		CONFIG : 'N U T, 0, 0, 0',
	X =  -84.898  mm,	Y =   -456.153  mm,	Z =   -229.176  mm,
	W =  90.000 deg,	P =   0.000 deg,	R =   90.000 deg
};
P[1878]{
   GP1:
	UF : 0, UT : 6,		CONFIG : 'N U T, 0, 0, 0',
	X =  -83.663  mm,	Y =   -458.430  mm,	Z =   -228.986  mm,
	W =  90.000 deg,	P =   0.000 deg,	R =   90.000 deg
};
P[1879]{
   GP1:
	UF : 0, UT : 6,		CONFIG : 'N U T, 0, 0, 0',
	X =  -82.928  mm,	Y =   -459.679  mm,	Z =   -229.020  mm,
	W =  90.000 deg,	P =   0.000 deg,	R =   90.000 deg
};
P[1880]{
   GP1:
	UF : 0, UT : 6,		CONFIG : 'N U T, 0, 0, 0',
	X =  -81.085  mm,	Y =   -462.911  mm,	Z =   -228.962  mm,
	W =  90.000 deg,	P =   0.000 deg,	R =   90.000 deg
};
P[1881]{
   GP1:
	UF : 0, UT : 6,		CONFIG : 'N U T, 0, 0, 0',
	X =  -80.232  mm,	Y =   -464.268  mm,	Z =   -229.131  mm,
	W =  90.000 deg,	P =   0.000 deg,	R =   90.000 deg
};
P[1882]{
   GP1:
	UF : 0, UT : 6,		CONFIG : 'N U T, 0, 0, 0',
	X =  -79.260  mm,	Y =   -465.944  mm,	Z =   -229.142  mm,
	W =  90.000 deg,	P =   0.000 deg,	R =   90.000 deg
};
P[1883]{
   GP1:
	UF : 0, UT : 6,		CONFIG : 'N U T, 0, 0, 0',
	X =  -78.133  mm,	Y =   -467.770  mm,	Z =   -229.317  mm,
	W =  90.000 deg,	P =   0.000 deg,	R =   90.000 deg
};
P[1884]{
   GP1:
	UF : 0, UT : 6,		CONFIG : 'N U T, 0, 0, 0',
	X =  -76.870  mm,	Y =   -470.008  mm,	Z =   -229.247  mm,
	W =  90.000 deg,	P =   0.000 deg,	R =   90.000 deg
};
P[1885]{
   GP1:
	UF : 0, UT : 6,		CONFIG : 'N U T, 0, 0, 0',
	X =  -76.601  mm,	Y =   -470.711  mm,	Z =   -228.915  mm,
	W =  90.000 deg,	P =   0.000 deg,	R =   90.000 deg
};
P[1886]{
   GP1:
	UF : 0, UT : 6,		CONFIG : 'N U T, 0, 0, 0',
	X =  -76.006  mm,	Y =   -471.663  mm,	Z =   -229.025  mm,
	W =  90.000 deg,	P =   0.000 deg,	R =   90.000 deg
};
P[1887]{
   GP1:
	UF : 0, UT : 6,		CONFIG : 'N U T, 0, 0, 0',
	X =  -75.413  mm,	Y =   -472.457  mm,	Z =   -229.353  mm,
	W =  90.000 deg,	P =   0.000 deg,	R =   90.000 deg
};
P[1888]{
   GP1:
	UF : 0, UT : 6,		CONFIG : 'N U T, 0, 0, 0',
	X =  -73.867  mm,	Y =   -475.295  mm,	Z =   -229.125  mm,
	W =  90.000 deg,	P =   0.000 deg,	R =   90.000 deg
};
P[1889]{
   GP1:
	UF : 0, UT : 6,		CONFIG : 'N U T, 0, 0, 0',
	X =  -73.257  mm,	Y =   -476.368  mm,	Z =   -229.103  mm,
	W =  90.000 deg,	P =   0.000 deg,	R =   90.000 deg
};
P[1890]{
   GP1:
	UF : 0, UT : 6,		CONFIG : 'N U T, 0, 0, 0',
	X =  -72.393  mm,	Y =   -477.925  mm,	Z =   -229.019  mm,
	W =  90.000 deg,	P =   0.000 deg,	R =   90.000 deg
};
P[1891]{
   GP1:
	UF : 0, UT : 6,		CONFIG : 'N U T, 0, 0, 0',
	X =  -70.648  mm,	Y =   -480.890  mm,	Z =   -229.099  mm,
	W =  90.000 deg,	P =   0.000 deg,	R =   90.000 deg
};
P[1892]{
   GP1:
	UF : 0, UT : 6,		CONFIG : 'N U T, 0, 0, 0',
	X =  -69.941  mm,	Y =   -482.226  mm,	Z =   -228.941  mm,
	W =  90.000 deg,	P =   0.000 deg,	R =   90.000 deg
};
P[1893]{
   GP1:
	UF : 0, UT : 6,		CONFIG : 'N U T, 0, 0, 0',
	X =  -68.745  mm,	Y =   -484.212  mm,	Z =   -229.061  mm,
	W =  90.000 deg,	P =   0.000 deg,	R =   90.000 deg
};
P[1894]{
   GP1:
	UF : 0, UT : 6,		CONFIG : 'N U T, 0, 0, 0',
	X =  -67.612  mm,	Y =   -486.179  mm,	Z =   -229.057  mm,
	W =  90.000 deg,	P =   0.000 deg,	R =   90.000 deg
};
P[1895]{
   GP1:
	UF : 0, UT : 6,		CONFIG : 'N U T, 0, 0, 0',
	X =  -67.186  mm,	Y =   -486.752  mm,	Z =   -229.286  mm,
	W =  90.000 deg,	P =   0.000 deg,	R =   90.000 deg
};
P[1896]{
   GP1:
	UF : 0, UT : 6,		CONFIG : 'N U T, 0, 0, 0',
	X =  -65.673  mm,	Y =   -489.345  mm,	Z =   -229.323  mm,
	W =  90.000 deg,	P =   0.000 deg,	R =   90.000 deg
};
P[1897]{
   GP1:
	UF : 0, UT : 6,		CONFIG : 'N U T, 0, 0, 0',
	X =  -64.016  mm,	Y =   -492.207  mm,	Z =   -229.338  mm,
	W =  90.000 deg,	P =   0.000 deg,	R =   90.000 deg
};
P[1898]{
   GP1:
	UF : 0, UT : 6,		CONFIG : 'N U T, 0, 0, 0',
	X =  -62.181  mm,	Y =   -495.525  mm,	Z =   -229.139  mm,
	W =  90.000 deg,	P =   0.000 deg,	R =   90.000 deg
};
P[1899]{
   GP1:
	UF : 0, UT : 6,		CONFIG : 'N U T, 0, 0, 0',
	X =  -61.771  mm,	Y =   -496.398  mm,	Z =   -228.910  mm,
	W =  90.000 deg,	P =   0.000 deg,	R =   90.000 deg
};
P[1900]{
   GP1:
	UF : 0, UT : 6,		CONFIG : 'N U T, 0, 0, 0',
	X =  -60.571  mm,	Y =   -498.326  mm,	Z =   -229.121  mm,
	W =  90.000 deg,	P =   0.000 deg,	R =   90.000 deg
};
P[1901]{
   GP1:
	UF : 0, UT : 6,		CONFIG : 'N U T, 0, 0, 0',
	X =  -59.881  mm,	Y =   -499.449  mm,	Z =   -229.224  mm,
	W =  90.000 deg,	P =   0.000 deg,	R =   90.000 deg
};
P[1902]{
   GP1:
	UF : 0, UT : 6,		CONFIG : 'N U T, 0, 0, 0',
	X =  -58.706  mm,	Y =   -501.474  mm,	Z =   -229.236  mm,
	W =  90.000 deg,	P =   0.000 deg,	R =   90.000 deg
};
P[1903]{
   GP1:
	UF : 0, UT : 6,		CONFIG : 'N U T, 0, 0, 0',
	X =  -57.602  mm,	Y =   -503.420  mm,	Z =   -229.192  mm,
	W =  90.000 deg,	P =   0.000 deg,	R =   90.000 deg
};
P[1904]{
   GP1:
	UF : 0, UT : 6,		CONFIG : 'N U T, 0, 0, 0',
	X =  -57.120  mm,	Y =   -504.223  mm,	Z =   -229.233  mm,
	W =  90.000 deg,	P =   0.000 deg,	R =   90.000 deg
};
P[1905]{
   GP1:
	UF : 0, UT : 6,		CONFIG : 'N U T, 0, 0, 0',
	X =  -56.073  mm,	Y =   -506.225  mm,	Z =   -228.970  mm,
	W =  90.000 deg,	P =   0.000 deg,	R =   90.000 deg
};
P[1906]{
   GP1:
	UF : 0, UT : 6,		CONFIG : 'N U T, 0, 0, 0',
	X =  -55.235  mm,	Y =   -507.685  mm,	Z =   -228.957  mm,
	W =  90.000 deg,	P =   0.000 deg,	R =   90.000 deg
};
P[1907]{
   GP1:
	UF : 0, UT : 6,		CONFIG : 'N U T, 0, 0, 0',
	X =  -54.533  mm,	Y =   -508.925  mm,	Z =   -228.924  mm,
	W =  90.000 deg,	P =   0.000 deg,	R =   90.000 deg
};
P[1908]{
   GP1:
	UF : 0, UT : 6,		CONFIG : 'N U T, 0, 0, 0',
	X =  -53.968  mm,	Y =   -509.842  mm,	Z =   -229.011  mm,
	W =  90.000 deg,	P =   0.000 deg,	R =   90.000 deg
};
P[1909]{
   GP1:
	UF : 0, UT : 6,		CONFIG : 'N U T, 0, 0, 0',
	X =  -52.733  mm,	Y =   -511.988  mm,	Z =   -229.001  mm,
	W =  90.000 deg,	P =   0.000 deg,	R =   90.000 deg
};
P[1910]{
   GP1:
	UF : 0, UT : 6,		CONFIG : 'N U T, 0, 0, 0',
	X =  -52.218  mm,	Y =   -512.794  mm,	Z =   -229.122  mm,
	W =  90.000 deg,	P =   0.000 deg,	R =   90.000 deg
};
P[1911]{
   GP1:
	UF : 0, UT : 6,		CONFIG : 'N U T, 0, 0, 0',
	X =  -51.448  mm,	Y =   -514.121  mm,	Z =   -229.130  mm,
	W =  90.000 deg,	P =   0.000 deg,	R =   90.000 deg
};
P[1912]{
   GP1:
	UF : 0, UT : 6,		CONFIG : 'N U T, 0, 0, 0',
	X =  -51.107  mm,	Y =   -514.734  mm,	Z =   -229.098  mm,
	W =  90.000 deg,	P =   0.000 deg,	R =   90.000 deg
};
P[1913]{
   GP1:
	UF : 0, UT : 6,		CONFIG : 'N U T, 0, 0, 0',
	X =  -50.400  mm,	Y =   -515.845  mm,	Z =   -229.257  mm,
	W =  90.000 deg,	P =   0.000 deg,	R =   90.000 deg
};
P[1914]{
   GP1:
	UF : 0, UT : 6,		CONFIG : 'N U T, 0, 0, 0',
	X =  -48.972  mm,	Y =   -518.526  mm,	Z =   -228.967  mm,
	W =  90.000 deg,	P =   0.000 deg,	R =   90.000 deg
};
P[1915]{
   GP1:
	UF : 0, UT : 6,		CONFIG : 'N U T, 0, 0, 0',
	X =  -48.636  mm,	Y =   -519.071  mm,	Z =   -229.017  mm,
	W =  90.000 deg,	P =   0.000 deg,	R =   90.000 deg
};
P[1916]{
   GP1:
	UF : 0, UT : 6,		CONFIG : 'N U T, 0, 0, 0',
	X =  -47.873  mm,	Y =   -520.244  mm,	Z =   -229.226  mm,
	W =  90.000 deg,	P =   0.000 deg,	R =   90.000 deg
};
P[1917]{
   GP1:
	UF : 0, UT : 6,		CONFIG : 'N U T, 0, 0, 0',
	X =  -47.615  mm,	Y =   -520.883  mm,	Z =   -228.958  mm,
	W =  90.000 deg,	P =   0.000 deg,	R =   90.000 deg
};
P[1918]{
   GP1:
	UF : 0, UT : 6,		CONFIG : 'N U T, 0, 0, 0',
	X =  -46.921  mm,	Y =   -521.821  mm,	Z =   -229.327  mm,
	W =  90.000 deg,	P =   0.000 deg,	R =   90.000 deg
};
P[1919]{
   GP1:
	UF : 0, UT : 6,		CONFIG : 'N U T, 0, 0, 0',
	X =  -46.013  mm,	Y =   -523.391  mm,	Z =   -229.328  mm,
	W =  90.000 deg,	P =   0.000 deg,	R =   90.000 deg
};
P[1920]{
   GP1:
	UF : 0, UT : 6,		CONFIG : 'N U T, 0, 0, 0',
	X =  -42.474  mm,	Y =   -529.727  mm,	Z =   -229.040  mm,
	W =  90.000 deg,	P =   0.000 deg,	R =   90.000 deg
};
P[1921]{
   GP1:
	UF : 0, UT : 6,		CONFIG : 'N U T, 0, 0, 0',
	X =  -42.047  mm,	Y =   -530.273  mm,	Z =   -229.311  mm,
	W =  90.000 deg,	P =   0.000 deg,	R =   90.000 deg
};
P[1922]{
   GP1:
	UF : 0, UT : 6,		CONFIG : 'N U T, 0, 0, 0',
	X =  -40.957  mm,	Y =   -532.439  mm,	Z =   -228.920  mm,
	W =  90.000 deg,	P =   0.000 deg,	R =   90.000 deg
};
P[1923]{
   GP1:
	UF : 0, UT : 6,		CONFIG : 'N U T, 0, 0, 0',
	X =  -40.136  mm,	Y =   -533.665  mm,	Z =   -229.195  mm,
	W =  90.000 deg,	P =   0.000 deg,	R =   90.000 deg
};
P[1924]{
   GP1:
	UF : 0, UT : 6,		CONFIG : 'N U T, 0, 0, 0',
	X =  -39.547  mm,	Y =   -534.548  mm,	Z =   -229.387  mm,
	W =  90.000 deg,	P =   0.000 deg,	R =   90.000 deg
};
P[1925]{
   GP1:
	UF : 0, UT : 6,		CONFIG : 'N U T, 0, 0, 0',
	X =  -39.111  mm,	Y =   -535.637  mm,	Z =   -228.922  mm,
	W =  90.000 deg,	P =   0.000 deg,	R =   90.000 deg
};
P[1926]{
   GP1:
	UF : 0, UT : 6,		CONFIG : 'N U T, 0, 0, 0',
	X =  -38.636  mm,	Y =   -536.139  mm,	Z =   -229.370  mm,
	W =  90.000 deg,	P =   0.000 deg,	R =   90.000 deg
};
P[1927]{
   GP1:
	UF : 0, UT : 6,		CONFIG : 'N U T, 0, 0, 0',
	X =  -37.772  mm,	Y =   -537.825  mm,	Z =   -229.103  mm,
	W =  90.000 deg,	P =   0.000 deg,	R =   90.000 deg
};
P[1928]{
   GP1:
	UF : 0, UT : 6,		CONFIG : 'N U T, 0, 0, 0',
	X =  -37.216  mm,	Y =   -538.618  mm,	Z =   -229.343  mm,
	W =  90.000 deg,	P =   0.000 deg,	R =   90.000 deg
};
P[1929]{
   GP1:
	UF : 0, UT : 6,		CONFIG : 'N U T, 0, 0, 0',
	X =  -36.840  mm,	Y =   -539.348  mm,	Z =   -229.232  mm,
	W =  90.000 deg,	P =   0.000 deg,	R =   90.000 deg
};
P[1930]{
   GP1:
	UF : 0, UT : 6,		CONFIG : 'N U T, 0, 0, 0',
	X =  -35.568  mm,	Y =   -541.606  mm,	Z =   -229.154  mm,
	W =  90.000 deg,	P =   0.000 deg,	R =   90.000 deg
};
P[1931]{
   GP1:
	UF : 0, UT : 6,		CONFIG : 'N U T, 0, 0, 0',
	X =  -34.214  mm,	Y =   -544.105  mm,	Z =   -228.940  mm,
	W =  90.000 deg,	P =   0.000 deg,	R =   90.000 deg
};
P[1932]{
   GP1:
	UF : 0, UT : 6,		CONFIG : 'N U T, 0, 0, 0',
	X =  -33.432  mm,	Y =   -545.291  mm,	Z =   -229.175  mm,
	W =  90.000 deg,	P =   0.000 deg,	R =   90.000 deg
};
P[1933]{
   GP1:
	UF : 0, UT : 6,		CONFIG : 'N U T, 0, 0, 0',
	X =  -33.013  mm,	Y =   -546.060  mm,	Z =   -229.112  mm,
	W =  90.000 deg,	P =   0.000 deg,	R =   90.000 deg
};
P[1934]{
   GP1:
	UF : 0, UT : 6,		CONFIG : 'N U T, 0, 0, 0',
	X =  -32.529  mm,	Y =   -547.015  mm,	Z =   -228.950  mm,
	W =  90.000 deg,	P =   0.000 deg,	R =   90.000 deg
};
P[1935]{
   GP1:
	UF : 0, UT : 6,		CONFIG : 'N U T, 0, 0, 0',
	X =  -31.449  mm,	Y =   -548.769  mm,	Z =   -229.114  mm,
	W =  90.000 deg,	P =   0.000 deg,	R =   90.000 deg
};
P[1936]{
   GP1:
	UF : 0, UT : 6,		CONFIG : 'N U T, 0, 0, 0',
	X =  -30.074  mm,	Y =   -551.151  mm,	Z =   -229.112  mm,
	W =  90.000 deg,	P =   0.000 deg,	R =   90.000 deg
};
P[1937]{
   GP1:
	UF : 0, UT : 6,		CONFIG : 'N U T, 0, 0, 0',
	X =  -29.313  mm,	Y =   -552.269  mm,	Z =   -229.394  mm,
	W =  90.000 deg,	P =   0.000 deg,	R =   90.000 deg
};
P[1938]{
   GP1:
	UF : 0, UT : 6,		CONFIG : 'N U T, 0, 0, 0',
	X =  -28.591  mm,	Y =   -553.768  mm,	Z =   -229.045  mm,
	W =  90.000 deg,	P =   0.000 deg,	R =   90.000 deg
};
P[1939]{
   GP1:
	UF : 0, UT : 6,		CONFIG : 'N U T, 0, 0, 0',
	X =  -28.197  mm,	Y =   -554.306  mm,	Z =   -229.246  mm,
	W =  90.000 deg,	P =   0.000 deg,	R =   90.000 deg
};
P[1940]{
   GP1:
	UF : 0, UT : 6,		CONFIG : 'N U T, 0, 0, 0',
	X =  -27.639  mm,	Y =   -555.385  mm,	Z =   -229.091  mm,
	W =  90.000 deg,	P =   0.000 deg,	R =   90.000 deg
};
P[1941]{
   GP1:
	UF : 0, UT : 6,		CONFIG : 'N U T, 0, 0, 0',
	X =  -27.305  mm,	Y =   -556.054  mm,	Z =   -228.961  mm,
	W =  90.000 deg,	P =   0.000 deg,	R =   90.000 deg
};
P[1942]{
   GP1:
	UF : 0, UT : 6,		CONFIG : 'N U T, 0, 0, 0',
	X =  -26.817  mm,	Y =   -556.750  mm,	Z =   -229.173  mm,
	W =  90.000 deg,	P =   0.000 deg,	R =   90.000 deg
};
P[1943]{
   GP1:
	UF : 0, UT : 6,		CONFIG : 'N U T, 0, 0, 0',
	X =  -26.448  mm,	Y =   -557.375  mm,	Z =   -229.192  mm,
	W =  90.000 deg,	P =   0.000 deg,	R =   90.000 deg
};
P[1944]{
   GP1:
	UF : 0, UT : 6,		CONFIG : 'N U T, 0, 0, 0',
	X =  -26.062  mm,	Y =   -557.913  mm,	Z =   -229.374  mm,
	W =  90.000 deg,	P =   0.000 deg,	R =   90.000 deg
};
P[1945]{
   GP1:
	UF : 0, UT : 6,		CONFIG : 'N U T, 0, 0, 0',
	X =  -25.445  mm,	Y =   -559.256  mm,	Z =   -228.990  mm,
	W =  90.000 deg,	P =   0.000 deg,	R =   90.000 deg
};
P[1946]{
   GP1:
	UF : 0, UT : 6,		CONFIG : 'N U T, 0, 0, 0',
	X =  -24.492  mm,	Y =   -560.881  mm,	Z =   -229.025  mm,
	W =  90.000 deg,	P =   0.000 deg,	R =   90.000 deg
};
P[1947]{
   GP1:
	UF : 0, UT : 6,		CONFIG : 'N U T, 0, 0, 0',
	X =  -24.115  mm,	Y =   -561.452  mm,	Z =   -229.142  mm,
	W =  90.000 deg,	P =   0.000 deg,	R =   90.000 deg
};
P[1948]{
   GP1:
	UF : 0, UT : 6,		CONFIG : 'N U T, 0, 0, 0',
	X =  -23.742  mm,	Y =   -562.033  mm,	Z =   -229.230  mm,
	W =  90.000 deg,	P =   0.000 deg,	R =   90.000 deg
};
P[1949]{
   GP1:
	UF : 0, UT : 6,		CONFIG : 'N U T, 0, 0, 0',
	X =  -23.239  mm,	Y =   -562.972  mm,	Z =   -229.137  mm,
	W =  90.000 deg,	P =   0.000 deg,	R =   90.000 deg
};
P[1950]{
   GP1:
	UF : 0, UT : 6,		CONFIG : 'N U T, 0, 0, 0',
	X =  -22.508  mm,	Y =   -564.173  mm,	Z =   -229.227  mm,
	W =  90.000 deg,	P =   0.000 deg,	R =   90.000 deg
};
P[1951]{
   GP1:
	UF : 0, UT : 6,		CONFIG : 'N U T, 0, 0, 0',
	X =  -22.225  mm,	Y =   -564.895  mm,	Z =   -228.903  mm,
	W =  90.000 deg,	P =   0.000 deg,	R =   90.000 deg
};
P[1952]{
   GP1:
	UF : 0, UT : 6,		CONFIG : 'N U T, 0, 0, 0',
	X =  -21.317  mm,	Y =   -566.450  mm,	Z =   -228.927  mm,
	W =  90.000 deg,	P =   0.000 deg,	R =   90.000 deg
};
P[1953]{
   GP1:
	UF : 0, UT : 6,		CONFIG : 'N U T, 0, 0, 0',
	X =  -20.255  mm,	Y =   -568.298  mm,	Z =   -228.915  mm,
	W =  90.000 deg,	P =   0.000 deg,	R =   90.000 deg
};
P[1954]{
   GP1:
	UF : 0, UT : 6,		CONFIG : 'N U T, 0, 0, 0',
	X =  -18.989  mm,	Y =   -570.230  mm,	Z =   -229.280  mm,
	W =  90.000 deg,	P =   0.000 deg,	R =   90.000 deg
};
P[1955]{
   GP1:
	UF : 0, UT : 6,		CONFIG : 'N U T, 0, 0, 0',
	X =  -18.050  mm,	Y =   -571.845  mm,	Z =   -229.296  mm,
	W =  90.000 deg,	P =   0.000 deg,	R =   90.000 deg
};
P[1956]{
   GP1:
	UF : 0, UT : 6,		CONFIG : 'N U T, 0, 0, 0',
	X =  -17.691  mm,	Y =   -572.466  mm,	Z =   -229.299  mm,
	W =  90.000 deg,	P =   0.000 deg,	R =   90.000 deg
};
P[1957]{
   GP1:
	UF : 0, UT : 6,		CONFIG : 'N U T, 0, 0, 0',
	X =  -15.916  mm,	Y =   -575.562  mm,	Z =   -229.268  mm,
	W =  90.000 deg,	P =   0.000 deg,	R =   90.000 deg
};
P[1958]{
   GP1:
	UF : 0, UT : 6,		CONFIG : 'N U T, 0, 0, 0',
	X =  -14.939  mm,	Y =   -577.378  mm,	Z =   -229.094  mm,
	W =  90.000 deg,	P =   0.000 deg,	R =   90.000 deg
};
P[1959]{
   GP1:
	UF : 0, UT : 6,		CONFIG : 'N U T, 0, 0, 0',
	X =  -13.601  mm,	Y =   -579.782  mm,	Z =   -228.974  mm,
	W =  90.000 deg,	P =   0.000 deg,	R =   90.000 deg
};
P[1960]{
   GP1:
	UF : 0, UT : 6,		CONFIG : 'N U T, 0, 0, 0',
	X =  -12.352  mm,	Y =   -581.982  mm,	Z =   -228.917  mm,
	W =  90.000 deg,	P =   0.000 deg,	R =   90.000 deg
};
P[1961]{
   GP1:
	UF : 0, UT : 6,		CONFIG : 'N U T, 0, 0, 0',
	X =  -10.773  mm,	Y =   -584.552  mm,	Z =   -229.149  mm,
	W =  90.000 deg,	P =   0.000 deg,	R =   90.000 deg
};
P[1962]{
   GP1:
	UF : 0, UT : 6,		CONFIG : 'N U T, 0, 0, 0',
	X =  -10.168  mm,	Y =   -585.526  mm,	Z =   -229.253  mm,
	W =  90.000 deg,	P =   0.000 deg,	R =   90.000 deg
};
P[1963]{
   GP1:
	UF : 0, UT : 6,		CONFIG : 'N U T, 0, 0, 0',
	X =  -9.050  mm,	Y =   -587.423  mm,	Z =   -229.308  mm,
	W =  90.000 deg,	P =   0.000 deg,	R =   90.000 deg
};
P[1964]{
   GP1:
	UF : 0, UT : 6,		CONFIG : 'N U T, 0, 0, 0',
	X =  -8.721  mm,	Y =   -588.247  mm,	Z =   -228.951  mm,
	W =  90.000 deg,	P =   0.000 deg,	R =   90.000 deg
};
P[1965]{
   GP1:
	UF : 0, UT : 6,		CONFIG : 'N U T, 0, 0, 0',
	X =  -7.932  mm,	Y =   -589.309  mm,	Z =   -229.380  mm,
	W =  90.000 deg,	P =   0.000 deg,	R =   90.000 deg
};
P[1966]{
   GP1:
	UF : 0, UT : 6,		CONFIG : 'N U T, 0, 0, 0',
	X =  -7.035  mm,	Y =   -590.953  mm,	Z =   -229.254  mm,
	W =  90.000 deg,	P =   0.000 deg,	R =   90.000 deg
};
P[1967]{
   GP1:
	UF : 0, UT : 6,		CONFIG : 'N U T, 0, 0, 0',
	X =  -6.081  mm,	Y =   -592.642  mm,	Z =   -229.200  mm,
	W =  90.000 deg,	P =   0.000 deg,	R =   90.000 deg
};
P[1968]{
   GP1:
	UF : 0, UT : 6,		CONFIG : 'N U T, 0, 0, 0',
	X =  -5.304  mm,	Y =   -593.877  mm,	Z =   -229.356  mm,
	W =  90.000 deg,	P =   0.000 deg,	R =   90.000 deg
};
P[1969]{
   GP1:
	UF : 0, UT : 6,		CONFIG : 'N U T, 0, 0, 0',
	X =  -2.340  mm,	Y =   -599.014  mm,	Z =   -229.351  mm,
	W =  90.000 deg,	P =   0.000 deg,	R =   90.000 deg
};
P[1970]{
   GP1:
	UF : 0, UT : 6,		CONFIG : 'N U T, 0, 0, 0',
	X =  -1.849  mm,	Y =   -599.941  mm,	Z =   -229.244  mm,
	W =  90.000 deg,	P =   0.000 deg,	R =   90.000 deg
};
P[1971]{
   GP1:
	UF : 0, UT : 6,		CONFIG : 'N U T, 0, 0, 0',
	X =  -0.825  mm,	Y =   -601.724  mm,	Z =   -229.231  mm,
	W =  90.000 deg,	P =   0.000 deg,	R =   90.000 deg
};
P[1972]{
   GP1:
	UF : 0, UT : 6,		CONFIG : 'N U T, 0, 0, 0',
	X =  1.170  mm,	Y =   -605.211  mm,	Z =   -229.186  mm,
	W =  90.000 deg,	P =   0.000 deg,	R =   90.000 deg
};
P[1973]{
   GP1:
	UF : 0, UT : 6,		CONFIG : 'N U T, 0, 0, 0',
	X =  2.075  mm,	Y =   -606.732  mm,	Z =   -229.252  mm,
	W =  90.000 deg,	P =   0.000 deg,	R =   90.000 deg
};
P[1974]{
   GP1:
	UF : 0, UT : 6,		CONFIG : 'N U T, 0, 0, 0',
	X =  2.429  mm,	Y =   -607.590  mm,	Z =   -228.907  mm,
	W =  90.000 deg,	P =   0.000 deg,	R =   90.000 deg
};
P[1975]{
   GP1:
	UF : 0, UT : 6,		CONFIG : 'N U T, 0, 0, 0',
	X =  3.314  mm,	Y =   -609.002  mm,	Z =   -229.077  mm,
	W =  90.000 deg,	P =   0.000 deg,	R =   90.000 deg
};
P[1976]{
   GP1:
	UF : 0, UT : 6,		CONFIG : 'N U T, 0, 0, 0',
	X =  4.028  mm,	Y =   -610.291  mm,	Z =   -229.004  mm,
	W =  90.000 deg,	P =   0.000 deg,	R =   90.000 deg
};
P[1977]{
   GP1:
	UF : 0, UT : 6,		CONFIG : 'N U T, 0, 0, 0',
	X =  5.234  mm,	Y =   -612.206  mm,	Z =   -229.248  mm,
	W =  90.000 deg,	P =   0.000 deg,	R =   90.000 deg
};
P[1978]{
   GP1:
	UF : 0, UT : 6,		CONFIG : 'N U T, 0, 0, 0',
	X =  6.128  mm,	Y =   -613.887  mm,	Z =   -229.062  mm,
	W =  90.000 deg,	P =   0.000 deg,	R =   90.000 deg
};
P[1979]{
   GP1:
	UF : 0, UT : 6,		CONFIG : 'N U T, 0, 0, 0',
	X =  6.614  mm,	Y =   -614.591  mm,	Z =   -229.254  mm,
	W =  90.000 deg,	P =   0.000 deg,	R =   90.000 deg
};
P[1980]{
   GP1:
	UF : 0, UT : 6,		CONFIG : 'N U T, 0, 0, 0',
	X =  7.020  mm,	Y =   -615.272  mm,	Z =   -229.285  mm,
	W =  90.000 deg,	P =   0.000 deg,	R =   90.000 deg
};
P[1981]{
   GP1:
	UF : 0, UT : 6,		CONFIG : 'N U T, 0, 0, 0',
	X =  7.653  mm,	Y =   -616.426  mm,	Z =   -229.207  mm,
	W =  90.000 deg,	P =   0.000 deg,	R =   90.000 deg
};
P[1982]{
   GP1:
	UF : 0, UT : 6,		CONFIG : 'N U T, 0, 0, 0',
	X =  10.100  mm,	Y =   -620.580  mm,	Z =   -229.323  mm,
	W =  90.000 deg,	P =   0.000 deg,	R =   90.000 deg
};
P[1983]{
   GP1:
	UF : 0, UT : 6,		CONFIG : 'N U T, 0, 0, 0',
	X =  11.139  mm,	Y =   -622.415  mm,	Z =   -229.274  mm,
	W =  90.000 deg,	P =   0.000 deg,	R =   90.000 deg
};
P[1984]{
   GP1:
	UF : 0, UT : 6,		CONFIG : 'N U T, 0, 0, 0',
	X =  12.419  mm,	Y =   -624.577  mm,	Z =   -229.349  mm,
	W =  90.000 deg,	P =   0.000 deg,	R =   90.000 deg
};
P[1985]{
   GP1:
	UF : 0, UT : 6,		CONFIG : 'N U T, 0, 0, 0',
	X =  14.477  mm,	Y =   -628.353  mm,	Z =   -229.055  mm,
	W =  90.000 deg,	P =   0.000 deg,	R =   90.000 deg
};
P[1986]{
   GP1:
	UF : 0, UT : 6,		CONFIG : 'N U T, 0, 0, 0',
	X =  15.195  mm,	Y =   -629.546  mm,	Z =   -229.123  mm,
	W =  90.000 deg,	P =   0.000 deg,	R =   90.000 deg
};
P[1987]{
   GP1:
	UF : 0, UT : 6,		CONFIG : 'N U T, 0, 0, 0',
	X =  16.393  mm,	Y =   -631.711  mm,	Z =   -228.998  mm,
	W =  90.000 deg,	P =   0.000 deg,	R =   90.000 deg
};
P[1988]{
   GP1:
	UF : 0, UT : 6,		CONFIG : 'N U T, 0, 0, 0',
	X =  18.034  mm,	Y =   -634.315  mm,	Z =   -229.331  mm,
	W =  90.000 deg,	P =   0.000 deg,	R =   90.000 deg
};
P[1989]{
   GP1:
	UF : 0, UT : 6,		CONFIG : 'N U T, 0, 0, 0',
	X =  18.392  mm,	Y =   -634.921  mm,	Z =   -229.350  mm,
	W =  90.000 deg,	P =   0.000 deg,	R =   90.000 deg
};
P[1990]{
   GP1:
	UF : 0, UT : 6,		CONFIG : 'N U T, 0, 0, 0',
	X =  20.159  mm,	Y =   -638.166  mm,	Z =   -229.092  mm,
	W =  90.000 deg,	P =   0.000 deg,	R =   90.000 deg
};
P[1991]{
   GP1:
	UF : 0, UT : 6,		CONFIG : 'N U T, 0, 0, 0',
	X =  20.589  mm,	Y =   -638.841  mm,	Z =   -229.191  mm,
	W =  90.000 deg,	P =   0.000 deg,	R =   90.000 deg
};
P[1992]{
   GP1:
	UF : 0, UT : 6,		CONFIG : 'N U T, 0, 0, 0',
	X =  21.020  mm,	Y =   -639.730  mm,	Z =   -228.990  mm,
	W =  90.000 deg,	P =   0.000 deg,	R =   90.000 deg
};
P[1993]{
   GP1:
	UF : 0, UT : 6,		CONFIG : 'N U T, 0, 0, 0',
	X =  21.635  mm,	Y =   -640.635  mm,	Z =   -229.213  mm,
	W =  90.000 deg,	P =   0.000 deg,	R =   90.000 deg
};
P[1994]{
   GP1:
	UF : 0, UT : 6,		CONFIG : 'N U T, 0, 0, 0',
	X =  22.551  mm,	Y =   -642.090  mm,	Z =   -229.398  mm,
	W =  90.000 deg,	P =   0.000 deg,	R =   90.000 deg
};
P[1995]{
   GP1:
	UF : 0, UT : 6,		CONFIG : 'N U T, 0, 0, 0',
	X =  23.720  mm,	Y =   -644.173  mm,	Z =   -229.317  mm,
	W =  90.000 deg,	P =   0.000 deg,	R =   90.000 deg
};
P[1996]{
   GP1:
	UF : 0, UT : 6,		CONFIG : 'N U T, 0, 0, 0',
	X =  23.992  mm,	Y =   -644.909  mm,	Z =   -228.945  mm,
	W =  90.000 deg,	P =   0.000 deg,	R =   90.000 deg
};
P[1997]{
   GP1:
	UF : 0, UT : 6,		CONFIG : 'N U T, 0, 0, 0',
	X =  24.458  mm,	Y =   -645.652  mm,	Z =   -229.037  mm,
	W =  90.000 deg,	P =   0.000 deg,	R =   90.000 deg
};
P[1998]{
   GP1:
	UF : 0, UT : 6,		CONFIG : 'N U T, 0, 0, 0',
	X =  26.461  mm,	Y =   -649.023  mm,	Z =   -229.172  mm,
	W =  90.000 deg,	P =   0.000 deg,	R =   90.000 deg
};
P[1999]{
   GP1:
	UF : 0, UT : 6,		CONFIG : 'N U T, 0, 0, 0',
	X =  27.064  mm,	Y =   -649.948  mm,	Z =   -229.339  mm,
	W =  90.000 deg,	P =   0.000 deg,	R =   90.000 deg
};
P[2000]{
   GP1:
	UF : 0, UT : 6,		CONFIG : 'N U T, 0, 0, 0',
	X =  28.968  mm,	Y =   -653.318  mm,	Z =   -229.240  mm,
	W =  90.000 deg,	P =   0.000 deg,	R =   90.000 deg
};
P[2001]{
   GP1:
	UF : 0, UT : 6,		CONFIG : 'N U T, 0, 0, 0',
	X =  29.240  mm,	Y =   -654.025  mm,	Z =   -228.908  mm,
	W =  90.000 deg,	P =   0.000 deg,	R =   90.000 deg
};
P[2002]{
   GP1:
	UF : 0, UT : 6,		CONFIG : 'N U T, 0, 0, 0',
	X =  30.326  mm,	Y =   -655.616  mm,	Z =   -229.313  mm,
	W =  90.000 deg,	P =   0.000 deg,	R =   90.000 deg
};
P[2003]{
   GP1:
	UF : 0, UT : 6,		CONFIG : 'N U T, 0, 0, 0',
	X =  30.854  mm,	Y =   -656.576  mm,	Z =   -229.250  mm,
	W =  90.000 deg,	P =   0.000 deg,	R =   90.000 deg
};
P[2004]{
   GP1:
	UF : 0, UT : 6,		CONFIG : 'N U T, 0, 0, 0',
	X =  31.658  mm,	Y =   -657.887  mm,	Z =   -229.364  mm,
	W =  90.000 deg,	P =   0.000 deg,	R =   90.000 deg
};
P[2005]{
   GP1:
	UF : 0, UT : 6,		CONFIG : 'N U T, 0, 0, 0',
	X =  31.929  mm,	Y =   -658.510  mm,	Z =   -229.151  mm,
	W =  90.000 deg,	P =   0.000 deg,	R =   90.000 deg
};
P[2006]{
   GP1:
	UF : 0, UT : 6,		CONFIG : 'N U T, 0, 0, 0',
	X =  32.203  mm,	Y =   -659.142  mm,	Z =   -228.927  mm,
	W =  90.000 deg,	P =   0.000 deg,	R =   90.000 deg
};
P[2007]{
   GP1:
	UF : 0, UT : 6,		CONFIG : 'N U T, 0, 0, 0',
	X =  33.215  mm,	Y =   -660.572  mm,	Z =   -229.381  mm,
	W =  90.000 deg,	P =   0.000 deg,	R =   90.000 deg
};
P[2008]{
   GP1:
	UF : 0, UT : 6,		CONFIG : 'N U T, 0, 0, 0',
	X =  33.684  mm,	Y =   -661.516  mm,	Z =   -229.196  mm,
	W =  90.000 deg,	P =   0.000 deg,	R =   90.000 deg
};
P[2009]{
   GP1:
	UF : 0, UT : 6,		CONFIG : 'N U T, 0, 0, 0',
	X =  34.084  mm,	Y =   -662.273  mm,	Z =   -229.106  mm,
	W =  90.000 deg,	P =   0.000 deg,	R =   90.000 deg
};
P[2010]{
   GP1:
	UF : 0, UT : 6,		CONFIG : 'N U T, 0, 0, 0',
	X =  34.657  mm,	Y =   -663.137  mm,	Z =   -229.284  mm,
	W =  90.000 deg,	P =   0.000 deg,	R =   90.000 deg
};
P[2011]{
   GP1:
	UF : 0, UT : 6,		CONFIG : 'N U T, 0, 0, 0',
	X =  35.348  mm,	Y =   -664.292  mm,	Z =   -229.345  mm,
	W =  90.000 deg,	P =   0.000 deg,	R =   90.000 deg
};
P[2012]{
   GP1:
	UF : 0, UT : 6,		CONFIG : 'N U T, 0, 0, 0',
	X =  35.814  mm,	Y =   -665.197  mm,	Z =   -229.207  mm,
	W =  90.000 deg,	P =   0.000 deg,	R =   90.000 deg
};
P[2013]{
   GP1:
	UF : 0, UT : 6,		CONFIG : 'N U T, 0, 0, 0',
	X =  36.114  mm,	Y =   -665.829  mm,	Z =   -229.050  mm,
	W =  90.000 deg,	P =   0.000 deg,	R =   90.000 deg
};
P[2014]{
   GP1:
	UF : 0, UT : 6,		CONFIG : 'N U T, 0, 0, 0',
	X =  37.039  mm,	Y =   -667.514  mm,	Z =   -228.935  mm,
	W =  90.000 deg,	P =   0.000 deg,	R =   90.000 deg
};
P[2015]{
   GP1:
	UF : 0, UT : 6,		CONFIG : 'N U T, 0, 0, 0',
	X =  37.980  mm,	Y =   -669.024  mm,	Z =   -229.100  mm,
	W =  90.000 deg,	P =   0.000 deg,	R =   90.000 deg
};
P[2016]{
   GP1:
	UF : 0, UT : 6,		CONFIG : 'N U T, 0, 0, 0',
	X =  38.312  mm,	Y =   -669.632  mm,	Z =   -229.055  mm,
	W =  90.000 deg,	P =   0.000 deg,	R =   90.000 deg
};
P[2017]{
   GP1:
	UF : 0, UT : 6,		CONFIG : 'N U T, 0, 0, 0',
	X =  39.131  mm,	Y =   -671.068  mm,	Z =   -229.028  mm,
	W =  90.000 deg,	P =   0.000 deg,	R =   90.000 deg
};
P[2018]{
   GP1:
	UF : 0, UT : 6,		CONFIG : 'N U T, 0, 0, 0',
	X =  40.632  mm,	Y =   -673.531  mm,	Z =   -229.221  mm,
	W =  90.000 deg,	P =   0.000 deg,	R =   90.000 deg
};
P[2019]{
   GP1:
	UF : 0, UT : 6,		CONFIG : 'N U T, 0, 0, 0',
	X =  41.052  mm,	Y =   -674.328  mm,	Z =   -229.124  mm,
	W =  90.000 deg,	P =   0.000 deg,	R =   90.000 deg
};
P[2020]{
   GP1:
	UF : 0, UT : 6,		CONFIG : 'N U T, 0, 0, 0',
	X =  41.680  mm,	Y =   -675.461  mm,	Z =   -229.058  mm,
	W =  90.000 deg,	P =   0.000 deg,	R =   90.000 deg
};
P[2021]{
   GP1:
	UF : 0, UT : 6,		CONFIG : 'N U T, 0, 0, 0',
	X =  42.038  mm,	Y =   -676.151  mm,	Z =   -228.961  mm,
	W =  90.000 deg,	P =   0.000 deg,	R =   90.000 deg
};
P[2022]{
   GP1:
	UF : 0, UT : 6,		CONFIG : 'N U T, 0, 0, 0',
	X =  43.636  mm,	Y =   -678.746  mm,	Z =   -229.206  mm,
	W =  90.000 deg,	P =   0.000 deg,	R =   90.000 deg
};
P[2023]{
   GP1:
	UF : 0, UT : 6,		CONFIG : 'N U T, 0, 0, 0',
	X =  45.042  mm,	Y =   -681.094  mm,	Z =   -229.326  mm,
	W =  90.000 deg,	P =   0.000 deg,	R =   90.000 deg
};
P[2024]{
   GP1:
	UF : 0, UT : 6,		CONFIG : 'N U T, 0, 0, 0',
	X =  45.971  mm,	Y =   -682.721  mm,	Z =   -229.126  mm,
	W =  90.000 deg,	P =   0.000 deg,	R =   90.000 deg
};
P[2025]{
   GP1:
	UF : 0, UT : 6,		CONFIG : 'N U T, 0, 0, 0',
	X =  49.022  mm,	Y =   -686.197  mm,	Z =   -228.966  mm,
	W =  90.000 deg,	P =   0.000 deg,	R =   90.000 deg
};
P[2026]{
   GP1:
	UF : 0, UT : 6,		CONFIG : 'N U T, 0, 0, 0',
	X =  50.459  mm,	Y =   -687.110  mm,	Z =   -229.029  mm,
	W =  90.000 deg,	P =   0.000 deg,	R =   90.000 deg
};
P[2027]{
   GP1:
	UF : 0, UT : 6,		CONFIG : 'N U T, 0, 0, 0',
	X =  51.959  mm,	Y =   -687.726  mm,	Z =   -229.231  mm,
	W =  90.000 deg,	P =   0.000 deg,	R =   90.000 deg
};
P[2028]{
   GP1:
	UF : 0, UT : 6,		CONFIG : 'N U T, 0, 0, 0',
	X =  52.825  mm,	Y =   -688.130  mm,	Z =   -229.080  mm,
	W =  90.000 deg,	P =   0.000 deg,	R =   90.000 deg
};
P[2029]{
   GP1:
	UF : 0, UT : 6,		CONFIG : 'N U T, 0, 0, 0',
	X =  54.225  mm,	Y =   -688.465  mm,	Z =   -229.122  mm,
	W =  90.000 deg,	P =   0.000 deg,	R =   90.000 deg
};
P[2030]{
   GP1:
	UF : 0, UT : 6,		CONFIG : 'N U T, 0, 0, 0',
	X =  57.057  mm,	Y =   -688.644  mm,	Z =   -229.192  mm,
	W =  90.000 deg,	P =   0.000 deg,	R =   90.000 deg
};
P[2031]{
   GP1:
	UF : 0, UT : 6,		CONFIG : 'N U T, 0, 0, 0',
	X =  60.328  mm,	Y =   -688.139  mm,	Z =   -229.129  mm,
	W =  90.000 deg,	P =   0.000 deg,	R =   90.000 deg
};
P[2032]{
   GP1:
	UF : 0, UT : 6,		CONFIG : 'N U T, 0, 0, 0',
	X =  61.379  mm,	Y =   -687.747  mm,	Z =   -229.167  mm,
	W =  90.000 deg,	P =   0.000 deg,	R =   90.000 deg
};
P[2033]{
   GP1:
	UF : 0, UT : 6,		CONFIG : 'N U T, 0, 0, 0',
	X =  61.973  mm,	Y =   -687.487  mm,	Z =   -229.143  mm,
	W =  90.000 deg,	P =   0.000 deg,	R =   90.000 deg
};
P[2034]{
   GP1:
	UF : 0, UT : 6,		CONFIG : 'N U T, 0, 0, 0',
	X =  63.283  mm,	Y =   -686.838  mm,	Z =   -229.250  mm,
	W =  90.000 deg,	P =   0.000 deg,	R =   90.000 deg
};
P[2035]{
   GP1:
	UF : 0, UT : 6,		CONFIG : 'N U T, 0, 0, 0',
	X =  64.612  mm,	Y =   -686.126  mm,	Z =   -229.114  mm,
	W =  90.000 deg,	P =   0.000 deg,	R =   90.000 deg
};
P[2036]{
   GP1:
	UF : 0, UT : 6,		CONFIG : 'N U T, 0, 0, 0',
	X =  67.708  mm,	Y =   -684.297  mm,	Z =   -229.216  mm,
	W =  90.000 deg,	P =   0.000 deg,	R =   90.000 deg
};
P[2037]{
   GP1:
	UF : 0, UT : 6,		CONFIG : 'N U T, 0, 0, 0',
	X =  70.853  mm,	Y =   -682.446  mm,	Z =   -229.302  mm,
	W =  90.000 deg,	P =   0.000 deg,	R =   90.000 deg
};
P[2038]{
   GP1:
	UF : 0, UT : 6,		CONFIG : 'N U T, 0, 0, 0',
	X =  72.458  mm,	Y =   -681.578  mm,	Z =   -229.158  mm,
	W =  90.000 deg,	P =   0.000 deg,	R =   90.000 deg
};
P[2039]{
   GP1:
	UF : 0, UT : 6,		CONFIG : 'N U T, 0, 0, 0',
	X =  73.714  mm,	Y =   -680.869  mm,	Z =   -229.118  mm,
	W =  90.000 deg,	P =   0.000 deg,	R =   90.000 deg
};
P[2040]{
   GP1:
	UF : 0, UT : 6,		CONFIG : 'N U T, 0, 0, 0',
	X =  74.973  mm,	Y =   -680.223  mm,	Z =   -228.924  mm,
	W =  90.000 deg,	P =   0.000 deg,	R =   90.000 deg
};
P[2041]{
   GP1:
	UF : 0, UT : 6,		CONFIG : 'N U T, 0, 0, 0',
	X =  77.994  mm,	Y =   -678.400  mm,	Z =   -229.113  mm,
	W =  90.000 deg,	P =   0.000 deg,	R =   90.000 deg
};
P[2042]{
   GP1:
	UF : 0, UT : 6,		CONFIG : 'N U T, 0, 0, 0',
	X =  78.542  mm,	Y =   -678.065  mm,	Z =   -229.159  mm,
	W =  90.000 deg,	P =   0.000 deg,	R =   90.000 deg
};
P[2043]{
   GP1:
	UF : 0, UT : 6,		CONFIG : 'N U T, 0, 0, 0',
	X =  79.970  mm,	Y =   -677.326  mm,	Z =   -228.952  mm,
	W =  90.000 deg,	P =   0.000 deg,	R =   90.000 deg
};
P[2044]{
   GP1:
	UF : 0, UT : 6,		CONFIG : 'N U T, 0, 0, 0',
	X =  81.489  mm,	Y =   -676.423  mm,	Z =   -229.013  mm,
	W =  90.000 deg,	P =   0.000 deg,	R =   90.000 deg
};
P[2045]{
   GP1:
	UF : 0, UT : 6,		CONFIG : 'N U T, 0, 0, 0',
	X =  82.302  mm,	Y =   -675.828  mm,	Z =   -229.318  mm,
	W =  90.000 deg,	P =   0.000 deg,	R =   90.000 deg
};
P[2046]{
   GP1:
	UF : 0, UT : 6,		CONFIG : 'N U T, 0, 0, 0',
	X =  83.509  mm,	Y =   -675.110  mm,	Z =   -229.370  mm,
	W =  90.000 deg,	P =   0.000 deg,	R =   90.000 deg
};
P[2047]{
   GP1:
	UF : 0, UT : 6,		CONFIG : 'N U T, 0, 0, 0',
	X =  84.455  mm,	Y =   -674.622  mm,	Z =   -229.229  mm,
	W =  90.000 deg,	P =   0.000 deg,	R =   90.000 deg
};
P[2048]{
   GP1:
	UF : 0, UT : 6,		CONFIG : 'N U T, 0, 0, 0',
	X =  85.570  mm,	Y =   -674.055  mm,	Z =   -229.042  mm,
	W =  90.000 deg,	P =   0.000 deg,	R =   90.000 deg
};
P[2049]{
   GP1:
	UF : 0, UT : 6,		CONFIG : 'N U T, 0, 0, 0',
	X =  88.333  mm,	Y =   -672.368  mm,	Z =   -229.265  mm,
	W =  90.000 deg,	P =   0.000 deg,	R =   90.000 deg
};
P[2050]{
   GP1:
	UF : 0, UT : 6,		CONFIG : 'N U T, 0, 0, 0',
	X =  91.664  mm,	Y =   -670.525  mm,	Z =   -229.069  mm,
	W =  90.000 deg,	P =   0.000 deg,	R =   90.000 deg
};
P[2051]{
   GP1:
	UF : 0, UT : 6,		CONFIG : 'N U T, 0, 0, 0',
	X =  92.854  mm,	Y =   -669.766  mm,	Z =   -229.243  mm,
	W =  90.000 deg,	P =   0.000 deg,	R =   90.000 deg
};
P[2052]{
   GP1:
	UF : 0, UT : 6,		CONFIG : 'N U T, 0, 0, 0',
	X =  93.565  mm,	Y =   -669.391  mm,	Z =   -229.157  mm,
	W =  90.000 deg,	P =   0.000 deg,	R =   90.000 deg
};
P[2053]{
   GP1:
	UF : 0, UT : 6,		CONFIG : 'N U T, 0, 0, 0',
	X =  94.370  mm,	Y =   -668.948  mm,	Z =   -229.102  mm,
	W =  90.000 deg,	P =   0.000 deg,	R =   90.000 deg
};
P[2054]{
   GP1:
	UF : 0, UT : 6,		CONFIG : 'N U T, 0, 0, 0',
	X =  95.074  mm,	Y =   -668.505  mm,	Z =   -229.193  mm,
	W =  90.000 deg,	P =   0.000 deg,	R =   90.000 deg
};
P[2055]{
   GP1:
	UF : 0, UT : 6,		CONFIG : 'N U T, 0, 0, 0',
	X =  95.632  mm,	Y =   -668.174  mm,	Z =   -229.214  mm,
	W =  90.000 deg,	P =   0.000 deg,	R =   90.000 deg
};
P[2056]{
   GP1:
	UF : 0, UT : 6,		CONFIG : 'N U T, 0, 0, 0',
	X =  98.296  mm,	Y =   -666.568  mm,	Z =   -229.380  mm,
	W =  90.000 deg,	P =   0.000 deg,	R =   90.000 deg
};
P[2057]{
   GP1:
	UF : 0, UT : 6,		CONFIG : 'N U T, 0, 0, 0',
	X =  99.335  mm,	Y =   -666.161  mm,	Z =   -228.909  mm,
	W =  90.000 deg,	P =   0.000 deg,	R =   90.000 deg
};
P[2058]{
   GP1:
	UF : 0, UT : 6,		CONFIG : 'N U T, 0, 0, 0',
	X =  101.467  mm,	Y =   -664.893  mm,	Z =   -229.001  mm,
	W =  90.000 deg,	P =   0.000 deg,	R =   90.000 deg
};
P[2059]{
   GP1:
	UF : 0, UT : 6,		CONFIG : 'N U T, 0, 0, 0',
	X =  104.289  mm,	Y =   -663.254  mm,	Z =   -229.023  mm,
	W =  90.000 deg,	P =   0.000 deg,	R =   90.000 deg
};
P[2060]{
   GP1:
	UF : 0, UT : 6,		CONFIG : 'N U T, 0, 0, 0',
	X =  108.061  mm,	Y =   -661.097  mm,	Z =   -228.974  mm,
	W =  90.000 deg,	P =   0.000 deg,	R =   90.000 deg
};
P[2061]{
   GP1:
	UF : 0, UT : 6,		CONFIG : 'N U T, 0, 0, 0',
	X =  110.425  mm,	Y =   -659.681  mm,	Z =   -229.097  mm,
	W =  90.000 deg,	P =   0.000 deg,	R =   90.000 deg
};
P[2062]{
   GP1:
	UF : 0, UT : 6,		CONFIG : 'N U T, 0, 0, 0',
	X =  113.002  mm,	Y =   -658.184  mm,	Z =   -229.120  mm,
	W =  90.000 deg,	P =   0.000 deg,	R =   90.000 deg
};
P[2063]{
   GP1:
	UF : 0, UT : 6,		CONFIG : 'N U T, 0, 0, 0',
	X =  114.075  mm,	Y =   -657.553  mm,	Z =   -229.147  mm,
	W =  90.000 deg,	P =   0.000 deg,	R =   90.000 deg
};
P[2064]{
   GP1:
	UF : 0, UT : 6,		CONFIG : 'N U T, 0, 0, 0',
	X =  115.059  mm,	Y =   -657.008  mm,	Z =   -229.091  mm,
	W =  90.000 deg,	P =   0.000 deg,	R =   90.000 deg
};
P[2065]{
   GP1:
	UF : 0, UT : 6,		CONFIG : 'N U T, 0, 0, 0',
	X =  116.034  mm,	Y =   -656.460  mm,	Z =   -229.055  mm,
	W =  90.000 deg,	P =   0.000 deg,	R =   90.000 deg
};
P[2066]{
   GP1:
	UF : 0, UT : 6,		CONFIG : 'N U T, 0, 0, 0',
	X =  116.760  mm,	Y =   -656.077  mm,	Z =   -228.967  mm,
	W =  90.000 deg,	P =   0.000 deg,	R =   90.000 deg
};
P[2067]{
   GP1:
	UF : 0, UT : 6,		CONFIG : 'N U T, 0, 0, 0',
	X =  117.411  mm,	Y =   -655.671  mm,	Z =   -229.039  mm,
	W =  90.000 deg,	P =   0.000 deg,	R =   90.000 deg
};
P[2068]{
   GP1:
	UF : 0, UT : 6,		CONFIG : 'N U T, 0, 0, 0',
	X =  124.789  mm,	Y =   -651.412  mm,	Z =   -229.036  mm,
	W =  90.000 deg,	P =   0.000 deg,	R =   90.000 deg
};
P[2069]{
   GP1:
	UF : 0, UT : 6,		CONFIG : 'N U T, 0, 0, 0',
	X =  125.677  mm,	Y =   -650.814  mm,	Z =   -229.245  mm,
	W =  90.000 deg,	P =   0.000 deg,	R =   90.000 deg
};
P[2070]{
   GP1:
	UF : 0, UT : 6,		CONFIG : 'N U T, 0, 0, 0',
	X =  127.724  mm,	Y =   -649.682  mm,	Z =   -229.124  mm,
	W =  90.000 deg,	P =   0.000 deg,	R =   90.000 deg
};
P[2071]{
   GP1:
	UF : 0, UT : 6,		CONFIG : 'N U T, 0, 0, 0',
	X =  128.466  mm,	Y =   -649.179  mm,	Z =   -229.305  mm,
	W =  90.000 deg,	P =   0.000 deg,	R =   90.000 deg
};
P[2072]{
   GP1:
	UF : 0, UT : 6,		CONFIG : 'N U T, 0, 0, 0',
	X =  129.442  mm,	Y =   -648.710  mm,	Z =   -229.075  mm,
	W =  90.000 deg,	P =   0.000 deg,	R =   90.000 deg
};
P[2073]{
   GP1:
	UF : 0, UT : 6,		CONFIG : 'N U T, 0, 0, 0',
	X =  132.294  mm,	Y =   -647.097  mm,	Z =   -228.992  mm,
	W =  90.000 deg,	P =   0.000 deg,	R =   90.000 deg
};
P[2074]{
   GP1:
	UF : 0, UT : 6,		CONFIG : 'N U T, 0, 0, 0',
	X =  133.145  mm,	Y =   -646.479  mm,	Z =   -229.302  mm,
	W =  90.000 deg,	P =   0.000 deg,	R =   90.000 deg
};
P[2075]{
   GP1:
	UF : 0, UT : 6,		CONFIG : 'N U T, 0, 0, 0',
	X =  134.559  mm,	Y =   -645.708  mm,	Z =   -229.189  mm,
	W =  90.000 deg,	P =   0.000 deg,	R =   90.000 deg
};
P[2076]{
   GP1:
	UF : 0, UT : 6,		CONFIG : 'N U T, 0, 0, 0',
	X =  135.517  mm,	Y =   -645.084  mm,	Z =   -229.362  mm,
	W =  90.000 deg,	P =   0.000 deg,	R =   90.000 deg
};
P[2077]{
   GP1:
	UF : 0, UT : 6,		CONFIG : 'N U T, 0, 0, 0',
	X =  136.145  mm,	Y =   -644.729  mm,	Z =   -229.344  mm,
	W =  90.000 deg,	P =   0.000 deg,	R =   90.000 deg
};
P[2078]{
   GP1:
	UF : 0, UT : 6,		CONFIG : 'N U T, 0, 0, 0',
	X =  137.540  mm,	Y =   -643.915  mm,	Z =   -229.365  mm,
	W =  90.000 deg,	P =   0.000 deg,	R =   90.000 deg
};
P[2079]{
   GP1:
	UF : 0, UT : 6,		CONFIG : 'N U T, 0, 0, 0',
	X =  140.726  mm,	Y =   -642.088  mm,	Z =   -229.336  mm,
	W =  90.000 deg,	P =   0.000 deg,	R =   90.000 deg
};
P[2080]{
   GP1:
	UF : 0, UT : 6,		CONFIG : 'N U T, 0, 0, 0',
	X =  142.026  mm,	Y =   -641.463  mm,	Z =   -229.029  mm,
	W =  90.000 deg,	P =   0.000 deg,	R =   90.000 deg
};
P[2081]{
   GP1:
	UF : 0, UT : 6,		CONFIG : 'N U T, 0, 0, 0',
	X =  143.527  mm,	Y =   -640.468  mm,	Z =   -229.341  mm,
	W =  90.000 deg,	P =   0.000 deg,	R =   90.000 deg
};
P[2082]{
   GP1:
	UF : 0, UT : 6,		CONFIG : 'N U T, 0, 0, 0',
	X =  144.688  mm,	Y =   -639.896  mm,	Z =   -229.100  mm,
	W =  90.000 deg,	P =   0.000 deg,	R =   90.000 deg
};
P[2083]{
   GP1:
	UF : 0, UT : 6,		CONFIG : 'N U T, 0, 0, 0',
	X =  145.856  mm,	Y =   -639.186  mm,	Z =   -229.186  mm,
	W =  90.000 deg,	P =   0.000 deg,	R =   90.000 deg
};
P[2084]{
   GP1:
	UF : 0, UT : 6,		CONFIG : 'N U T, 0, 0, 0',
	X =  146.506  mm,	Y =   -638.726  mm,	Z =   -229.392  mm,
	W =  90.000 deg,	P =   0.000 deg,	R =   90.000 deg
};
P[2085]{
   GP1:
	UF : 0, UT : 6,		CONFIG : 'N U T, 0, 0, 0',
	X =  147.580  mm,	Y =   -638.260  mm,	Z =   -229.019  mm,
	W =  90.000 deg,	P =   0.000 deg,	R =   90.000 deg
};
P[2086]{
   GP1:
	UF : 0, UT : 6,		CONFIG : 'N U T, 0, 0, 0',
	X =  149.343  mm,	Y =   -637.179  mm,	Z =   -229.173  mm,
	W =  90.000 deg,	P =   0.000 deg,	R =   90.000 deg
};
P[2087]{
   GP1:
	UF : 0, UT : 6,		CONFIG : 'N U T, 0, 0, 0',
	X =  150.060  mm,	Y =   -636.866  mm,	Z =   -228.928  mm,
	W =  90.000 deg,	P =   0.000 deg,	R =   90.000 deg
};
P[2088]{
   GP1:
	UF : 0, UT : 6,		CONFIG : 'N U T, 0, 0, 0',
	X =  151.906  mm,	Y =   -635.664  mm,	Z =   -229.258  mm,
	W =  90.000 deg,	P =   0.000 deg,	R =   90.000 deg
};
P[2089]{
   GP1:
	UF : 0, UT : 6,		CONFIG : 'N U T, 0, 0, 0',
	X =  153.935  mm,	Y =   -634.610  mm,	Z =   -228.972  mm,
	W =  90.000 deg,	P =   0.000 deg,	R =   90.000 deg
};
P[2090]{
   GP1:
	UF : 0, UT : 6,		CONFIG : 'N U T, 0, 0, 0',
	X =  155.249  mm,	Y =   -633.757  mm,	Z =   -229.200  mm,
	W =  90.000 deg,	P =   0.000 deg,	R =   90.000 deg
};
P[2091]{
   GP1:
	UF : 0, UT : 6,		CONFIG : 'N U T, 0, 0, 0',
	X =  157.657  mm,	Y =   -632.427  mm,	Z =   -229.055  mm,
	W =  90.000 deg,	P =   0.000 deg,	R =   90.000 deg
};
P[2092]{
   GP1:
	UF : 0, UT : 6,		CONFIG : 'N U T, 0, 0, 0',
	X =  158.686  mm,	Y =   -631.769  mm,	Z =   -229.210  mm,
	W =  90.000 deg,	P =   0.000 deg,	R =   90.000 deg
};
P[2093]{
   GP1:
	UF : 0, UT : 6,		CONFIG : 'N U T, 0, 0, 0',
	X =  159.289  mm,	Y =   -631.512  mm,	Z =   -228.987  mm,
	W =  90.000 deg,	P =   0.000 deg,	R =   90.000 deg
};
P[2094]{
   GP1:
	UF : 0, UT : 6,		CONFIG : 'N U T, 0, 0, 0',
	X =  159.916  mm,	Y =   -631.000  mm,	Z =   -229.353  mm,
	W =  90.000 deg,	P =   0.000 deg,	R =   90.000 deg
};
P[2095]{
   GP1:
	UF : 0, UT : 6,		CONFIG : 'N U T, 0, 0, 0',
	X =  162.117  mm,	Y =   -629.793  mm,	Z =   -229.199  mm,
	W =  90.000 deg,	P =   0.000 deg,	R =   90.000 deg
};
P[2096]{
   GP1:
	UF : 0, UT : 6,		CONFIG : 'N U T, 0, 0, 0',
	X =  166.309  mm,	Y =   -627.421  mm,	Z =   -229.079  mm,
	W =  90.000 deg,	P =   0.000 deg,	R =   90.000 deg
};
P[2097]{
   GP1:
	UF : 0, UT : 6,		CONFIG : 'N U T, 0, 0, 0',
	X =  169.311  mm,	Y =   -625.581  mm,	Z =   -229.340  mm,
	W =  90.000 deg,	P =   0.000 deg,	R =   90.000 deg
};
P[2098]{
   GP1:
	UF : 0, UT : 6,		CONFIG : 'N U T, 0, 0, 0',
	X =  173.100  mm,	Y =   -623.478  mm,	Z =   -229.134  mm,
	W =  90.000 deg,	P =   0.000 deg,	R =   90.000 deg
};
P[2099]{
   GP1:
	UF : 0, UT : 6,		CONFIG : 'N U T, 0, 0, 0',
	X =  175.148  mm,	Y =   -622.316  mm,	Z =   -229.085  mm,
	W =  90.000 deg,	P =   0.000 deg,	R =   90.000 deg
};
P[2100]{
   GP1:
	UF : 0, UT : 6,		CONFIG : 'N U T, 0, 0, 0',
	X =  177.450  mm,	Y =   -621.034  mm,	Z =   -228.971  mm,
	W =  90.000 deg,	P =   0.000 deg,	R =   90.000 deg
};
P[2101]{
   GP1:
	UF : 0, UT : 6,		CONFIG : 'N U T, 0, 0, 0',
	X =  178.437  mm,	Y =   -620.477  mm,	Z =   -228.938  mm,
	W =  90.000 deg,	P =   0.000 deg,	R =   90.000 deg
};
P[2102]{
   GP1:
	UF : 0, UT : 6,		CONFIG : 'N U T, 0, 0, 0',
	X =  179.159  mm,	Y =   -620.063  mm,	Z =   -228.930  mm,
	W =  90.000 deg,	P =   0.000 deg,	R =   90.000 deg
};
P[2103]{
   GP1:
	UF : 0, UT : 6,		CONFIG : 'N U T, 0, 0, 0',
	X =  180.551  mm,	Y =   -619.209  mm,	Z =   -229.051  mm,
	W =  90.000 deg,	P =   0.000 deg,	R =   90.000 deg
};
P[2104]{
   GP1:
	UF : 0, UT : 6,		CONFIG : 'N U T, 0, 0, 0',
	X =  181.818  mm,	Y =   -618.431  mm,	Z =   -229.167  mm,
	W =  90.000 deg,	P =   0.000 deg,	R =   90.000 deg
};
P[2105]{
   GP1:
	UF : 0, UT : 6,		CONFIG : 'N U T, 0, 0, 0',
	X =  183.298  mm,	Y =   -617.500  mm,	Z =   -229.352  mm,
	W =  90.000 deg,	P =   0.000 deg,	R =   90.000 deg
};
P[2106]{
   GP1:
	UF : 0, UT : 6,		CONFIG : 'N U T, 0, 0, 0',
	X =  184.271  mm,	Y =   -617.052  mm,	Z =   -229.076  mm,
	W =  90.000 deg,	P =   0.000 deg,	R =   90.000 deg
};
P[2107]{
   GP1:
	UF : 0, UT : 6,		CONFIG : 'N U T, 0, 0, 0',
	X =  187.137  mm,	Y =   -615.400  mm,	Z =   -229.070  mm,
	W =  90.000 deg,	P =   0.000 deg,	R =   90.000 deg
};
P[2108]{
   GP1:
	UF : 0, UT : 6,		CONFIG : 'N U T, 0, 0, 0',
	X =  188.418  mm,	Y =   -614.682  mm,	Z =   -229.016  mm,
	W =  90.000 deg,	P =   0.000 deg,	R =   90.000 deg
};
P[2109]{
   GP1:
	UF : 0, UT : 6,		CONFIG : 'N U T, 0, 0, 0',
	X =  189.566  mm,	Y =   -614.000  mm,	Z =   -229.062  mm,
	W =  90.000 deg,	P =   0.000 deg,	R =   90.000 deg
};
P[2110]{
   GP1:
	UF : 0, UT : 6,		CONFIG : 'N U T, 0, 0, 0',
	X =  191.235  mm,	Y =   -613.103  mm,	Z =   -228.901  mm,
	W =  90.000 deg,	P =   0.000 deg,	R =   90.000 deg
};
P[2111]{
   GP1:
	UF : 0, UT : 6,		CONFIG : 'N U T, 0, 0, 0',
	X =  195.420  mm,	Y =   -610.528  mm,	Z =   -229.286  mm,
	W =  90.000 deg,	P =   0.000 deg,	R =   90.000 deg
};
P[2112]{
   GP1:
	UF : 0, UT : 6,		CONFIG : 'N U T, 0, 0, 0',
	X =  198.504  mm,	Y =   -608.792  mm,	Z =   -229.178  mm,
	W =  90.000 deg,	P =   0.000 deg,	R =   90.000 deg
};
P[2113]{
   GP1:
	UF : 0, UT : 6,		CONFIG : 'N U T, 0, 0, 0',
	X =  199.088  mm,	Y =   -608.408  mm,	Z =   -229.292  mm,
	W =  90.000 deg,	P =   0.000 deg,	R =   90.000 deg
};
P[2114]{
   GP1:
	UF : 0, UT : 6,		CONFIG : 'N U T, 0, 0, 0',
	X =  200.227  mm,	Y =   -607.866  mm,	Z =   -229.010  mm,
	W =  90.000 deg,	P =   0.000 deg,	R =   90.000 deg
};
P[2115]{
   GP1:
	UF : 0, UT : 6,		CONFIG : 'N U T, 0, 0, 0',
	X =  203.674  mm,	Y =   -605.864  mm,	Z =   -229.038  mm,
	W =  90.000 deg,	P =   0.000 deg,	R =   90.000 deg
};
P[2116]{
   GP1:
	UF : 0, UT : 6,		CONFIG : 'N U T, 0, 0, 0',
	X =  204.445  mm,	Y =   -605.349  mm,	Z =   -229.208  mm,
	W =  90.000 deg,	P =   0.000 deg,	R =   90.000 deg
};
P[2117]{
   GP1:
	UF : 0, UT : 6,		CONFIG : 'N U T, 0, 0, 0',
	X =  206.842  mm,	Y =   -603.937  mm,	Z =   -229.275  mm,
	W =  90.000 deg,	P =   0.000 deg,	R =   90.000 deg
};
P[2118]{
   GP1:
	UF : 0, UT : 6,		CONFIG : 'N U T, 0, 0, 0',
	X =  207.468  mm,	Y =   -603.617  mm,	Z =   -229.176  mm,
	W =  90.000 deg,	P =   0.000 deg,	R =   90.000 deg
};
P[2119]{
   GP1:
	UF : 0, UT : 6,		CONFIG : 'N U T, 0, 0, 0',
	X =  208.757  mm,	Y =   -602.927  mm,	Z =   -229.045  mm,
	W =  90.000 deg,	P =   0.000 deg,	R =   90.000 deg
};
P[2120]{
   GP1:
	UF : 0, UT : 6,		CONFIG : 'N U T, 0, 0, 0',
	X =  209.478  mm,	Y =   -602.518  mm,	Z =   -229.026  mm,
	W =  90.000 deg,	P =   0.000 deg,	R =   90.000 deg
};
P[2121]{
   GP1:
	UF : 0, UT : 6,		CONFIG : 'N U T, 0, 0, 0',
	X =  210.909  mm,	Y =   -601.673  mm,	Z =   -229.071  mm,
	W =  90.000 deg,	P =   0.000 deg,	R =   90.000 deg
};
P[2122]{
   GP1:
	UF : 0, UT : 6,		CONFIG : 'N U T, 0, 0, 0',
	X =  211.779  mm,	Y =   -601.214  mm,	Z =   -228.966  mm,
	W =  90.000 deg,	P =   0.000 deg,	R =   90.000 deg
};
P[2123]{
   GP1:
	UF : 0, UT : 6,		CONFIG : 'N U T, 0, 0, 0',
	X =  212.720  mm,	Y =   -600.654  mm,	Z =   -229.007  mm,
	W =  90.000 deg,	P =   0.000 deg,	R =   90.000 deg
};
P[2124]{
   GP1:
	UF : 0, UT : 6,		CONFIG : 'N U T, 0, 0, 0',
	X =  213.728  mm,	Y =   -600.088  mm,	Z =   -228.967  mm,
	W =  90.000 deg,	P =   0.000 deg,	R =   90.000 deg
};
P[2125]{
   GP1:
	UF : 0, UT : 6,		CONFIG : 'N U T, 0, 0, 0',
	X =  217.187  mm,	Y =   -598.092  mm,	Z =   -228.965  mm,
	W =  90.000 deg,	P =   0.000 deg,	R =   90.000 deg
};
P[2126]{
   GP1:
	UF : 0, UT : 6,		CONFIG : 'N U T, 0, 0, 0',
	X =  218.715  mm,	Y =   -597.170  mm,	Z =   -229.062  mm,
	W =  90.000 deg,	P =   0.000 deg,	R =   90.000 deg
};
P[2127]{
   GP1:
	UF : 0, UT : 6,		CONFIG : 'N U T, 0, 0, 0',
	X =  220.918  mm,	Y =   -595.832  mm,	Z =   -229.222  mm,
	W =  90.000 deg,	P =   0.000 deg,	R =   90.000 deg
};
P[2128]{
   GP1:
	UF : 0, UT : 6,		CONFIG : 'N U T, 0, 0, 0',
	X =  222.796  mm,	Y =   -594.816  mm,	Z =   -229.055  mm,
	W =  90.000 deg,	P =   0.000 deg,	R =   90.000 deg
};
P[2129]{
   GP1:
	UF : 0, UT : 6,		CONFIG : 'N U T, 0, 0, 0',
	X =  223.457  mm,	Y =   -594.399  mm,	Z =   -229.142  mm,
	W =  90.000 deg,	P =   0.000 deg,	R =   90.000 deg
};
P[2130]{
   GP1:
	UF : 0, UT : 6,		CONFIG : 'N U T, 0, 0, 0',
	X =  224.224  mm,	Y =   -593.870  mm,	Z =   -229.351  mm,
	W =  90.000 deg,	P =   0.000 deg,	R =   90.000 deg
};
P[2131]{
   GP1:
	UF : 0, UT : 6,		CONFIG : 'N U T, 0, 0, 0',
	X =  226.075  mm,	Y =   -592.842  mm,	Z =   -229.253  mm,
	W =  90.000 deg,	P =   0.000 deg,	R =   90.000 deg
};
P[2132]{
   GP1:
	UF : 0, UT : 6,		CONFIG : 'N U T, 0, 0, 0',
	X =  226.918  mm,	Y =   -592.473  mm,	Z =   -228.966  mm,
	W =  90.000 deg,	P =   0.000 deg,	R =   90.000 deg
};
P[2133]{
   GP1:
	UF : 0, UT : 6,		CONFIG : 'N U T, 0, 0, 0',
	X =  227.767  mm,	Y =   -591.975  mm,	Z =   -228.986  mm,
	W =  90.000 deg,	P =   0.000 deg,	R =   90.000 deg
};
P[2134]{
   GP1:
	UF : 0, UT : 6,		CONFIG : 'N U T, 0, 0, 0',
	X =  228.339  mm,	Y =   -591.557  mm,	Z =   -229.199  mm,
	W =  90.000 deg,	P =   0.000 deg,	R =   90.000 deg
};
P[2135]{
   GP1:
	UF : 0, UT : 6,		CONFIG : 'N U T, 0, 0, 0',
	X =  231.154  mm,	Y =   -589.983  mm,	Z =   -229.077  mm,
	W =  90.000 deg,	P =   0.000 deg,	R =   90.000 deg
};
P[2136]{
   GP1:
	UF : 0, UT : 6,		CONFIG : 'N U T, 0, 0, 0',
	X =  231.832  mm,	Y =   -589.576  mm,	Z =   -229.110  mm,
	W =  90.000 deg,	P =   0.000 deg,	R =   90.000 deg
};
P[2137]{
   GP1:
	UF : 0, UT : 6,		CONFIG : 'N U T, 0, 0, 0',
	X =  233.678  mm,	Y =   -588.431  mm,	Z =   -229.305  mm,
	W =  90.000 deg,	P =   0.000 deg,	R =   90.000 deg
};
P[2138]{
   GP1:
	UF : 0, UT : 6,		CONFIG : 'N U T, 0, 0, 0',
	X =  235.936  mm,	Y =   -587.231  mm,	Z =   -229.053  mm,
	W =  90.000 deg,	P =   0.000 deg,	R =   90.000 deg
};
P[2139]{
   GP1:
	UF : 0, UT : 6,		CONFIG : 'N U T, 0, 0, 0',
	X =  237.170  mm,	Y =   -586.574  mm,	Z =   -228.915  mm,
	W =  90.000 deg,	P =   0.000 deg,	R =   90.000 deg
};
P[2140]{
   GP1:
	UF : 0, UT : 6,		CONFIG : 'N U T, 0, 0, 0',
	X =  240.266  mm,	Y =   -584.662  mm,	Z =   -229.219  mm,
	W =  90.000 deg,	P =   0.000 deg,	R =   90.000 deg
};
P[2141]{
   GP1:
	UF : 0, UT : 6,		CONFIG : 'N U T, 0, 0, 0',
	X =  240.916  mm,	Y =   -584.406  mm,	Z =   -228.928  mm,
	W =  90.000 deg,	P =   0.000 deg,	R =   90.000 deg
};
P[2142]{
   GP1:
	UF : 0, UT : 6,		CONFIG : 'N U T, 0, 0, 0',
	X =  241.542  mm,	Y =   -583.885  mm,	Z =   -229.316  mm,
	W =  90.000 deg,	P =   0.000 deg,	R =   90.000 deg
};
P[2143]{
   GP1:
	UF : 0, UT : 6,		CONFIG : 'N U T, 0, 0, 0',
	X =  242.391  mm,	Y =   -583.466  mm,	Z =   -229.145  mm,
	W =  90.000 deg,	P =   0.000 deg,	R =   90.000 deg
};
P[2144]{
   GP1:
	UF : 0, UT : 6,		CONFIG : 'N U T, 0, 0, 0',
	X =  243.227  mm,	Y =   -582.931  mm,	Z =   -229.270  mm,
	W =  90.000 deg,	P =   0.000 deg,	R =   90.000 deg
};
P[2145]{
   GP1:
	UF : 0, UT : 6,		CONFIG : 'N U T, 0, 0, 0',
	X =  244.471  mm,	Y =   -582.202  mm,	Z =   -229.297  mm,
	W =  90.000 deg,	P =   0.000 deg,	R =   90.000 deg
};
P[2146]{
   GP1:
	UF : 0, UT : 6,		CONFIG : 'N U T, 0, 0, 0',
	X =  247.592  mm,	Y =   -580.447  mm,	Z =   -229.184  mm,
	W =  90.000 deg,	P =   0.000 deg,	R =   90.000 deg
};
P[2147]{
   GP1:
	UF : 0, UT : 6,		CONFIG : 'N U T, 0, 0, 0',
	X =  250.336  mm,	Y =   -578.775  mm,	Z =   -229.394  mm,
	W =  90.000 deg,	P =   0.000 deg,	R =   90.000 deg
};
P[2148]{
   GP1:
	UF : 0, UT : 6,		CONFIG : 'N U T, 0, 0, 0',
	X =  251.843  mm,	Y =   -578.021  mm,	Z =   -229.114  mm,
	W =  90.000 deg,	P =   0.000 deg,	R =   90.000 deg
};
P[2149]{
   GP1:
	UF : 0, UT : 6,		CONFIG : 'N U T, 0, 0, 0',
	X =  252.752  mm,	Y =   -577.532  mm,	Z =   -229.026  mm,
	W =  90.000 deg,	P =   0.000 deg,	R =   90.000 deg
};
P[2150]{
   GP1:
	UF : 0, UT : 6,		CONFIG : 'N U T, 0, 0, 0',
	X =  255.224  mm,	Y =   -576.131  mm,	Z =   -228.961  mm,
	W =  90.000 deg,	P =   0.000 deg,	R =   90.000 deg
};
P[2151]{
   GP1:
	UF : 0, UT : 6,		CONFIG : 'N U T, 0, 0, 0',
	X =  256.407  mm,	Y =   -575.375  mm,	Z =   -229.139  mm,
	W =  90.000 deg,	P =   0.000 deg,	R =   90.000 deg
};
P[2152]{
   GP1:
	UF : 0, UT : 6,		CONFIG : 'N U T, 0, 0, 0',
	X =  257.819  mm,	Y =   -574.514  mm,	Z =   -229.248  mm,
	W =  90.000 deg,	P =   0.000 deg,	R =   90.000 deg
};
P[2153]{
   GP1:
	UF : 0, UT : 6,		CONFIG : 'N U T, 0, 0, 0',
	X =  259.952  mm,	Y =   -573.410  mm,	Z =   -228.942  mm,
	W =  90.000 deg,	P =   0.000 deg,	R =   90.000 deg
};
P[2154]{
   GP1:
	UF : 0, UT : 6,		CONFIG : 'N U T, 0, 0, 0',
	X =  261.091  mm,	Y =   -572.634  mm,	Z =   -229.229  mm,
	W =  90.000 deg,	P =   0.000 deg,	R =   90.000 deg
};
P[2155]{
   GP1:
	UF : 0, UT : 6,		CONFIG : 'N U T, 0, 0, 0',
	X =  262.801  mm,	Y =   -571.770  mm,	Z =   -228.928  mm,
	W =  90.000 deg,	P =   0.000 deg,	R =   90.000 deg
};
P[2156]{
   GP1:
	UF : 0, UT : 6,		CONFIG : 'N U T, 0, 0, 0',
	X =  263.888  mm,	Y =   -571.128  mm,	Z =   -228.962  mm,
	W =  90.000 deg,	P =   0.000 deg,	R =   90.000 deg
};
P[2157]{
   GP1:
	UF : 0, UT : 6,		CONFIG : 'N U T, 0, 0, 0',
	X =  266.470  mm,	Y =   -569.614  mm,	Z =   -229.019  mm,
	W =  90.000 deg,	P =   0.000 deg,	R =   90.000 deg
};
P[2158]{
   GP1:
	UF : 0, UT : 6,		CONFIG : 'N U T, 0, 0, 0',
	X =  268.589  mm,	Y =   -568.388  mm,	Z =   -229.025  mm,
	W =  90.000 deg,	P =   0.000 deg,	R =   90.000 deg
};
P[2159]{
   GP1:
	UF : 0, UT : 6,		CONFIG : 'N U T, 0, 0, 0',
	X =  271.619  mm,	Y =   -566.644  mm,	Z =   -229.013  mm,
	W =  90.000 deg,	P =   0.000 deg,	R =   90.000 deg
};
P[2160]{
   GP1:
	UF : 0, UT : 6,		CONFIG : 'N U T, 0, 0, 0',
	X =  273.105  mm,	Y =   -565.635  mm,	Z =   -229.381  mm,
	W =  90.000 deg,	P =   0.000 deg,	R =   90.000 deg
};
P[2161]{
   GP1:
	UF : 0, UT : 6,		CONFIG : 'N U T, 0, 0, 0',
	X =  276.067  mm,	Y =   -563.970  mm,	Z =   -229.269  mm,
	W =  90.000 deg,	P =   0.000 deg,	R =   90.000 deg
};
P[2162]{
   GP1:
	UF : 0, UT : 6,		CONFIG : 'N U T, 0, 0, 0',
	X =  280.768  mm,	Y =   -561.297  mm,	Z =   -229.168  mm,
	W =  90.000 deg,	P =   0.000 deg,	R =   90.000 deg
};
P[2163]{
   GP1:
	UF : 0, UT : 6,		CONFIG : 'N U T, 0, 0, 0',
	X =  281.698  mm,	Y =   -560.704  mm,	Z =   -229.305  mm,
	W =  90.000 deg,	P =   0.000 deg,	R =   90.000 deg
};
P[2164]{
   GP1:
	UF : 0, UT : 6,		CONFIG : 'N U T, 0, 0, 0',
	X =  282.741  mm,	Y =   -560.211  mm,	Z =   -229.038  mm,
	W =  90.000 deg,	P =   0.000 deg,	R =   90.000 deg
};
P[2165]{
   GP1:
	UF : 0, UT : 6,		CONFIG : 'N U T, 0, 0, 0',
	X =  283.543  mm,	Y =   -559.717  mm,	Z =   -229.113  mm,
	W =  90.000 deg,	P =   0.000 deg,	R =   90.000 deg
};
P[2166]{
   GP1:
	UF : 0, UT : 6,		CONFIG : 'N U T, 0, 0, 0',
	X =  286.790  mm,	Y =   -557.863  mm,	Z =   -229.064  mm,
	W =  90.000 deg,	P =   0.000 deg,	R =   90.000 deg
};
P[2167]{
   GP1:
	UF : 0, UT : 6,		CONFIG : 'N U T, 0, 0, 0',
	X =  288.201  mm,	Y =   -556.982  mm,	Z =   -229.224  mm,
	W =  90.000 deg,	P =   0.000 deg,	R =   90.000 deg
};
P[2168]{
   GP1:
	UF : 0, UT : 6,		CONFIG : 'N U T, 0, 0, 0',
	X =  288.885  mm,	Y =   -556.722  mm,	Z =   -228.899  mm,
	W =  90.000 deg,	P =   0.000 deg,	R =   90.000 deg
};
P[2169]{
   GP1:
	UF : 0, UT : 6,		CONFIG : 'N U T, 0, 0, 0',
	X =  289.966  mm,	Y =   -556.009  mm,	Z =   -229.113  mm,
	W =  90.000 deg,	P =   0.000 deg,	R =   90.000 deg
};
P[2170]{
   GP1:
	UF : 0, UT : 6,		CONFIG : 'N U T, 0, 0, 0',
	X =  291.800  mm,	Y =   -555.030  mm,	Z =   -228.919  mm,
	W =  90.000 deg,	P =   0.000 deg,	R =   90.000 deg
};
P[2171]{
   GP1:
	UF : 0, UT : 6,		CONFIG : 'N U T, 0, 0, 0',
	X =  292.753  mm,	Y =   -554.404  mm,	Z =   -229.102  mm,
	W =  90.000 deg,	P =   0.000 deg,	R =   90.000 deg
};
P[2172]{
   GP1:
	UF : 0, UT : 6,		CONFIG : 'N U T, 0, 0, 0',
	X =  293.257  mm,	Y =   -554.009  mm,	Z =   -229.355  mm,
	W =  90.000 deg,	P =   0.000 deg,	R =   90.000 deg
};
P[2173]{
   GP1:
	UF : 0, UT : 6,		CONFIG : 'N U T, 0, 0, 0',
	X =  295.081  mm,	Y =   -552.938  mm,	Z =   -229.397  mm,
	W =  90.000 deg,	P =   0.000 deg,	R =   90.000 deg
};
P[2174]{
   GP1:
	UF : 0, UT : 6,		CONFIG : 'N U T, 0, 0, 0',
	X =  296.168  mm,	Y =   -552.358  mm,	Z =   -229.283  mm,
	W =  90.000 deg,	P =   0.000 deg,	R =   90.000 deg
};
P[2175]{
   GP1:
	UF : 0, UT : 6,		CONFIG : 'N U T, 0, 0, 0',
	X =  296.875  mm,	Y =   -552.005  mm,	Z =   -229.149  mm,
	W =  90.000 deg,	P =   0.000 deg,	R =   90.000 deg
};
P[2176]{
   GP1:
	UF : 0, UT : 6,		CONFIG : 'N U T, 0, 0, 0',
	X =  297.991  mm,	Y =   -551.346  mm,	Z =   -229.186  mm,
	W =  90.000 deg,	P =   0.000 deg,	R =   90.000 deg
};
P[2177]{
   GP1:
	UF : 0, UT : 6,		CONFIG : 'N U T, 0, 0, 0',
	X =  300.674  mm,	Y =   -549.896  mm,	Z =   -228.943  mm,
	W =  90.000 deg,	P =   0.000 deg,	R =   90.000 deg
};
P[2178]{
   GP1:
	UF : 0, UT : 6,		CONFIG : 'N U T, 0, 0, 0',
	X =  302.278  mm,	Y =   -548.790  mm,	Z =   -229.381  mm,
	W =  90.000 deg,	P =   0.000 deg,	R =   90.000 deg
};
P[2179]{
   GP1:
	UF : 0, UT : 6,		CONFIG : 'N U T, 0, 0, 0',
	X =  304.654  mm,	Y =   -547.531  mm,	Z =   -229.108  mm,
	W =  90.000 deg,	P =   0.000 deg,	R =   90.000 deg
};
P[2180]{
   GP1:
	UF : 0, UT : 6,		CONFIG : 'N U T, 0, 0, 0',
	X =  305.308  mm,	Y =   -547.213  mm,	Z =   -228.963  mm,
	W =  90.000 deg,	P =   0.000 deg,	R =   90.000 deg
};
P[2181]{
   GP1:
	UF : 0, UT : 6,		CONFIG : 'N U T, 0, 0, 0',
	X =  306.887  mm,	Y =   -546.129  mm,	Z =   -229.380  mm,
	W =  90.000 deg,	P =   0.000 deg,	R =   90.000 deg
};
P[2182]{
   GP1:
	UF : 0, UT : 6,		CONFIG : 'N U T, 0, 0, 0',
	X =  307.570  mm,	Y =   -545.901  mm,	Z =   -228.977  mm,
	W =  90.000 deg,	P =   0.000 deg,	R =   90.000 deg
};
P[2183]{
   GP1:
	UF : 0, UT : 6,		CONFIG : 'N U T, 0, 0, 0',
	X =  309.996  mm,	Y =   -544.432  mm,	Z =   -229.141  mm,
	W =  90.000 deg,	P =   0.000 deg,	R =   90.000 deg
};
P[2184]{
   GP1:
	UF : 0, UT : 6,		CONFIG : 'N U T, 0, 0, 0',
	X =  310.638  mm,	Y =   -544.001  mm,	Z =   -229.287  mm,
	W =  90.000 deg,	P =   0.000 deg,	R =   90.000 deg
};
P[2185]{
   GP1:
	UF : 0, UT : 6,		CONFIG : 'N U T, 0, 0, 0',
	X =  312.328  mm,	Y =   -543.065  mm,	Z =   -229.189  mm,
	W =  90.000 deg,	P =   0.000 deg,	R =   90.000 deg
};
P[2186]{
   GP1:
	UF : 0, UT : 6,		CONFIG : 'N U T, 0, 0, 0',
	X =  314.247  mm,	Y =   -542.010  mm,	Z =   -229.062  mm,
	W =  90.000 deg,	P =   0.000 deg,	R =   90.000 deg
};
P[2187]{
   GP1:
	UF : 0, UT : 6,		CONFIG : 'N U T, 0, 0, 0',
	X =  315.101  mm,	Y =   -541.404  mm,	Z =   -229.338  mm,
	W =  90.000 deg,	P =   0.000 deg,	R =   90.000 deg
};
P[2188]{
   GP1:
	UF : 0, UT : 6,		CONFIG : 'N U T, 0, 0, 0',
	X =  316.750  mm,	Y =   -540.429  mm,	Z =   -229.392  mm,
	W =  90.000 deg,	P =   0.000 deg,	R =   90.000 deg
};
P[2189]{
   GP1:
	UF : 0, UT : 6,		CONFIG : 'N U T, 0, 0, 0',
	X =  317.275  mm,	Y =   -540.279  mm,	Z =   -229.020  mm,
	W =  90.000 deg,	P =   0.000 deg,	R =   90.000 deg
};
P[2190]{
   GP1:
	UF : 0, UT : 6,		CONFIG : 'N U T, 0, 0, 0',
	X =  320.616  mm,	Y =   -538.242  mm,	Z =   -229.283  mm,
	W =  90.000 deg,	P =   0.000 deg,	R =   90.000 deg
};
P[2191]{
   GP1:
	UF : 0, UT : 6,		CONFIG : 'N U T, 0, 0, 0',
	X =  322.579  mm,	Y =   -537.239  mm,	Z =   -228.966  mm,
	W =  90.000 deg,	P =   0.000 deg,	R =   90.000 deg
};
P[2192]{
   GP1:
	UF : 0, UT : 6,		CONFIG : 'N U T, 0, 0, 0',
	X =  327.038  mm,	Y =   -534.550  mm,	Z =   -229.244  mm,
	W =  90.000 deg,	P =   0.000 deg,	R =   90.000 deg
};
P[2193]{
   GP1:
	UF : 0, UT : 6,		CONFIG : 'N U T, 0, 0, 0',
	X =  327.589  mm,	Y =   -534.358  mm,	Z =   -228.939  mm,
	W =  90.000 deg,	P =   0.000 deg,	R =   90.000 deg
};
P[2194]{
   GP1:
	UF : 0, UT : 6,		CONFIG : 'N U T, 0, 0, 0',
	X =  328.726  mm,	Y =   -533.523  mm,	Z =   -229.372  mm,
	W =  90.000 deg,	P =   0.000 deg,	R =   90.000 deg
};
P[2195]{
   GP1:
	UF : 0, UT : 6,		CONFIG : 'N U T, 0, 0, 0',
	X =  331.617  mm,	Y =   -532.032  mm,	Z =   -228.938  mm,
	W =  90.000 deg,	P =   0.000 deg,	R =   90.000 deg
};
P[2196]{
   GP1:
	UF : 0, UT : 6,		CONFIG : 'N U T, 0, 0, 0',
	X =  334.454  mm,	Y =   -530.273  mm,	Z =   -229.232  mm,
	W =  90.000 deg,	P =   0.000 deg,	R =   90.000 deg
};
P[2197]{
   GP1:
	UF : 0, UT : 6,		CONFIG : 'N U T, 0, 0, 0',
	X =  336.870  mm,	Y =   -528.816  mm,	Z =   -229.384  mm,
	W =  90.000 deg,	P =   0.000 deg,	R =   90.000 deg
};
P[2198]{
   GP1:
	UF : 0, UT : 6,		CONFIG : 'N U T, 0, 0, 0',
	X =  338.100  mm,	Y =   -528.172  mm,	Z =   -229.221  mm,
	W =  90.000 deg,	P =   0.000 deg,	R =   90.000 deg
};
P[2199]{
   GP1:
	UF : 0, UT : 6,		CONFIG : 'N U T, 0, 0, 0',
	X =  339.434  mm,	Y =   -527.521  mm,	Z =   -228.934  mm,
	W =  90.000 deg,	P =   0.000 deg,	R =   90.000 deg
};
P[2200]{
   GP1:
	UF : 0, UT : 6,		CONFIG : 'N U T, 0, 0, 0',
	X =  343.787  mm,	Y =   -524.986  mm,	Z =   -228.986  mm,
	W =  90.000 deg,	P =   0.000 deg,	R =   90.000 deg
};
P[2201]{
   GP1:
	UF : 0, UT : 6,		CONFIG : 'N U T, 0, 0, 0',
	X =  346.111  mm,	Y =   -523.636  mm,	Z =   -229.006  mm,
	W =  90.000 deg,	P =   0.000 deg,	R =   90.000 deg
};
P[2202]{
   GP1:
	UF : 0, UT : 6,		CONFIG : 'N U T, 0, 0, 0',
	X =  351.106  mm,	Y =   -520.635  mm,	Z =   -229.288  mm,
	W =  90.000 deg,	P =   0.000 deg,	R =   90.000 deg
};
P[2203]{
   GP1:
	UF : 0, UT : 6,		CONFIG : 'N U T, 0, 0, 0',
	X =  352.238  mm,	Y =   -519.992  mm,	Z =   -229.262  mm,
	W =  90.000 deg,	P =   0.000 deg,	R =   90.000 deg
};
P[2204]{
   GP1:
	UF : 0, UT : 6,		CONFIG : 'N U T, 0, 0, 0',
	X =  354.086  mm,	Y =   -518.959  mm,	Z =   -229.179  mm,
	W =  90.000 deg,	P =   0.000 deg,	R =   90.000 deg
};
P[2205]{
   GP1:
	UF : 0, UT : 6,		CONFIG : 'N U T, 0, 0, 0',
	X =  356.460  mm,	Y =   -517.657  mm,	Z =   -229.014  mm,
	W =  90.000 deg,	P =   0.000 deg,	R =   90.000 deg
};
P[2206]{
   GP1:
	UF : 0, UT : 6,		CONFIG : 'N U T, 0, 0, 0',
	X =  356.865  mm,	Y =   -517.266  mm,	Z =   -229.396  mm,
	W =  90.000 deg,	P =   0.000 deg,	R =   90.000 deg
};
P[2207]{
   GP1:
	UF : 0, UT : 6,		CONFIG : 'N U T, 0, 0, 0',
	X =  357.565  mm,	Y =   -516.920  mm,	Z =   -229.254  mm,
	W =  90.000 deg,	P =   0.000 deg,	R =   90.000 deg
};
P[2208]{
   GP1:
	UF : 0, UT : 6,		CONFIG : 'N U T, 0, 0, 0',
	X =  359.182  mm,	Y =   -516.118  mm,	Z =   -228.933  mm,
	W =  90.000 deg,	P =   0.000 deg,	R =   90.000 deg
};
P[2209]{
   GP1:
	UF : 0, UT : 6,		CONFIG : 'N U T, 0, 0, 0',
	X =  361.003  mm,	Y =   -514.941  mm,	Z =   -229.240  mm,
	W =  90.000 deg,	P =   0.000 deg,	R =   90.000 deg
};
P[2210]{
   GP1:
	UF : 0, UT : 6,		CONFIG : 'N U T, 0, 0, 0',
	X =  362.302  mm,	Y =   -514.206  mm,	Z =   -229.203  mm,
	W =  90.000 deg,	P =   0.000 deg,	R =   90.000 deg
};
P[2211]{
   GP1:
	UF : 0, UT : 6,		CONFIG : 'N U T, 0, 0, 0',
	X =  363.483  mm,	Y =   -513.453  mm,	Z =   -229.375  mm,
	W =  90.000 deg,	P =   0.000 deg,	R =   90.000 deg
};
P[2212]{
   GP1:
	UF : 0, UT : 6,		CONFIG : 'N U T, 0, 0, 0',
	X =  364.830  mm,	Y =   -512.702  mm,	Z =   -229.311  mm,
	W =  90.000 deg,	P =   0.000 deg,	R =   90.000 deg
};
P[2213]{
   GP1:
	UF : 0, UT : 6,		CONFIG : 'N U T, 0, 0, 0',
	X =  365.913  mm,	Y =   -512.055  mm,	Z =   -229.362  mm,
	W =  90.000 deg,	P =   0.000 deg,	R =   90.000 deg
};
P[2214]{
   GP1:
	UF : 0, UT : 6,		CONFIG : 'N U T, 0, 0, 0',
	X =  366.534  mm,	Y =   -511.865  mm,	Z =   -228.954  mm,
	W =  90.000 deg,	P =   0.000 deg,	R =   90.000 deg
};
P[2215]{
   GP1:
	UF : 0, UT : 6,		CONFIG : 'N U T, 0, 0, 0',
	X =  367.230  mm,	Y =   -511.471  mm,	Z =   -228.936  mm,
	W =  90.000 deg,	P =   0.000 deg,	R =   90.000 deg
};
P[2216]{
   GP1:
	UF : 0, UT : 6,		CONFIG : 'N U T, 0, 0, 0',
	X =  367.828  mm,	Y =   -511.125  mm,	Z =   -228.936  mm,
	W =  90.000 deg,	P =   0.000 deg,	R =   90.000 deg
};
P[2217]{
   GP1:
	UF : 0, UT : 6,		CONFIG : 'N U T, 0, 0, 0',
	X =  368.313  mm,	Y =   -510.713  mm,	Z =   -229.259  mm,
	W =  90.000 deg,	P =   0.000 deg,	R =   90.000 deg
};
P[2218]{
   GP1:
	UF : 0, UT : 6,		CONFIG : 'N U T, 0, 0, 0',
	X =  369.998  mm,	Y =   -509.708  mm,	Z =   -229.334  mm,
	W =  90.000 deg,	P =   0.000 deg,	R =   90.000 deg
};
P[2219]{
   GP1:
	UF : 0, UT : 6,		CONFIG : 'N U T, 0, 0, 0',
	X =  370.542  mm,	Y =   -509.548  mm,	Z =   -228.958  mm,
	W =  90.000 deg,	P =   0.000 deg,	R =   90.000 deg
};
P[2220]{
   GP1:
	UF : 0, UT : 6,		CONFIG : 'N U T, 0, 0, 0',
	X =  371.034  mm,	Y =   -509.109  mm,	Z =   -229.337  mm,
	W =  90.000 deg,	P =   0.000 deg,	R =   90.000 deg
};
P[2221]{
   GP1:
	UF : 0, UT : 6,		CONFIG : 'N U T, 0, 0, 0',
	X =  371.746  mm,	Y =   -508.828  mm,	Z =   -229.021  mm,
	W =  90.000 deg,	P =   0.000 deg,	R =   90.000 deg
};
P[2222]{
   GP1:
	UF : 0, UT : 6,		CONFIG : 'N U T, 0, 0, 0',
	X =  372.397  mm,	Y =   -508.342  mm,	Z =   -229.288  mm,
	W =  90.000 deg,	P =   0.000 deg,	R =   90.000 deg
};
P[2223]{
   GP1:
	UF : 0, UT : 6,		CONFIG : 'N U T, 0, 0, 0',
	X =  375.558  mm,	Y =   -506.516  mm,	Z =   -229.291  mm,
	W =  90.000 deg,	P =   0.000 deg,	R =   90.000 deg
};
P[2224]{
   GP1:
	UF : 0, UT : 6,		CONFIG : 'N U T, 0, 0, 0',
	X =  376.745  mm,	Y =   -505.919  mm,	Z =   -229.078  mm,
	W =  90.000 deg,	P =   0.000 deg,	R =   90.000 deg
};
P[2225]{
   GP1:
	UF : 0, UT : 6,		CONFIG : 'N U T, 0, 0, 0',
	X =  378.767  mm,	Y =   -504.651  mm,	Z =   -229.320  mm,
	W =  90.000 deg,	P =   0.000 deg,	R =   90.000 deg
};
P[2226]{
   GP1:
	UF : 0, UT : 6,		CONFIG : 'N U T, 0, 0, 0',
	X =  381.304  mm,	Y =   -503.290  mm,	Z =   -229.066  mm,
	W =  90.000 deg,	P =   0.000 deg,	R =   90.000 deg
};
P[2227]{
   GP1:
	UF : 0, UT : 6,		CONFIG : 'N U T, 0, 0, 0',
	X =  383.850  mm,	Y =   -501.867  mm,	Z =   -228.956  mm,
	W =  90.000 deg,	P =   0.000 deg,	R =   90.000 deg
};
P[2228]{
   GP1:
	UF : 0, UT : 6,		CONFIG : 'N U T, 0, 0, 0',
	X =  386.398  mm,	Y =   -500.246  mm,	Z =   -229.316  mm,
	W =  90.000 deg,	P =   0.000 deg,	R =   90.000 deg
};
P[2229]{
   GP1:
	UF : 0, UT : 6,		CONFIG : 'N U T, 0, 0, 0',
	X =  387.632  mm,	Y =   -499.610  mm,	Z =   -229.131  mm,
	W =  90.000 deg,	P =   0.000 deg,	R =   90.000 deg
};
P[2230]{
   GP1:
	UF : 0, UT : 6,		CONFIG : 'N U T, 0, 0, 0',
	X =  390.135  mm,	Y =   -498.082  mm,	Z =   -229.330  mm,
	W =  90.000 deg,	P =   0.000 deg,	R =   90.000 deg
};
P[2231]{
   GP1:
	UF : 0, UT : 6,		CONFIG : 'N U T, 0, 0, 0',
	X =  390.913  mm,	Y =   -497.796  mm,	Z =   -228.937  mm,
	W =  90.000 deg,	P =   0.000 deg,	R =   90.000 deg
};
P[2232]{
   GP1:
	UF : 0, UT : 6,		CONFIG : 'N U T, 0, 0, 0',
	X =  393.186  mm,	Y =   -496.483  mm,	Z =   -228.936  mm,
	W =  90.000 deg,	P =   0.000 deg,	R =   90.000 deg
};
P[2233]{
   GP1:
	UF : 0, UT : 6,		CONFIG : 'N U T, 0, 0, 0',
	X =  395.387  mm,	Y =   -495.204  mm,	Z =   -228.956  mm,
	W =  90.000 deg,	P =   0.000 deg,	R =   90.000 deg
};
P[2234]{
   GP1:
	UF : 0, UT : 6,		CONFIG : 'N U T, 0, 0, 0',
	X =  396.200  mm,	Y =   -494.561  mm,	Z =   -229.378  mm,
	W =  90.000 deg,	P =   0.000 deg,	R =   90.000 deg
};
P[2235]{
   GP1:
	UF : 0, UT : 6,		CONFIG : 'N U T, 0, 0, 0',
	X =  398.494  mm,	Y =   -493.377  mm,	Z =   -229.040  mm,
	W =  90.000 deg,	P =   0.000 deg,	R =   90.000 deg
};
P[2236]{
   GP1:
	UF : 0, UT : 6,		CONFIG : 'N U T, 0, 0, 0',
	X =  399.012  mm,	Y =   -492.998  mm,	Z =   -229.232  mm,
	W =  90.000 deg,	P =   0.000 deg,	R =   90.000 deg
};
P[2237]{
   GP1:
	UF : 0, UT : 6,		CONFIG : 'N U T, 0, 0, 0',
	X =  400.780  mm,	Y =   -491.939  mm,	Z =   -229.324  mm,
	W =  90.000 deg,	P =   0.000 deg,	R =   90.000 deg
};
P[2238]{
   GP1:
	UF : 0, UT : 6,		CONFIG : 'N U T, 0, 0, 0',
	X =  404.136  mm,	Y =   -490.141  mm,	Z =   -228.986  mm,
	W =  90.000 deg,	P =   0.000 deg,	R =   90.000 deg
};
P[2239]{
   GP1:
	UF : 0, UT : 6,		CONFIG : 'N U T, 0, 0, 0',
	X =  406.982  mm,	Y =   -488.499  mm,	Z =   -228.981  mm,
	W =  90.000 deg,	P =   0.000 deg,	R =   90.000 deg
};
P[2240]{
   GP1:
	UF : 0, UT : 6,		CONFIG : 'N U T, 0, 0, 0',
	X =  408.951  mm,	Y =   -487.316  mm,	Z =   -229.092  mm,
	W =  90.000 deg,	P =   0.000 deg,	R =   90.000 deg
};
P[2241]{
   GP1:
	UF : 0, UT : 6,		CONFIG : 'N U T, 0, 0, 0',
	X =  409.637  mm,	Y =   -486.857  mm,	Z =   -229.247  mm,
	W =  90.000 deg,	P =   0.000 deg,	R =   90.000 deg
};
P[2242]{
   GP1:
	UF : 0, UT : 6,		CONFIG : 'N U T, 0, 0, 0',
	X =  413.728  mm,	Y =   -484.560  mm,	Z =   -229.088  mm,
	W =  90.000 deg,	P =   0.000 deg,	R =   90.000 deg
};
P[2243]{
   GP1:
	UF : 0, UT : 6,		CONFIG : 'N U T, 0, 0, 0',
	X =  415.865  mm,	Y =   -483.302  mm,	Z =   -229.145  mm,
	W =  90.000 deg,	P =   0.000 deg,	R =   90.000 deg
};
P[2244]{
   GP1:
	UF : 0, UT : 6,		CONFIG : 'N U T, 0, 0, 0',
	X =  416.680  mm,	Y =   -482.830  mm,	Z =   -229.151  mm,
	W =  90.000 deg,	P =   0.000 deg,	R =   90.000 deg
};
P[2245]{
   GP1:
	UF : 0, UT : 6,		CONFIG : 'N U T, 0, 0, 0',
	X =  419.255  mm,	Y =   -481.375  mm,	Z =   -229.075  mm,
	W =  90.000 deg,	P =   0.000 deg,	R =   90.000 deg
};
P[2246]{
   GP1:
	UF : 0, UT : 6,		CONFIG : 'N U T, 0, 0, 0',
	X =  420.269  mm,	Y =   -480.674  mm,	Z =   -229.353  mm,
	W =  90.000 deg,	P =   0.000 deg,	R =   90.000 deg
};
P[2247]{
   GP1:
	UF : 0, UT : 6,		CONFIG : 'N U T, 0, 0, 0',
	X =  422.574  mm,	Y =   -479.530  mm,	Z =   -228.901  mm,
	W =  90.000 deg,	P =   0.000 deg,	R =   90.000 deg
};
P[2248]{
   GP1:
	UF : 0, UT : 6,		CONFIG : 'N U T, 0, 0, 0',
	X =  424.629  mm,	Y =   -478.332  mm,	Z =   -228.928  mm,
	W =  90.000 deg,	P =   0.000 deg,	R =   90.000 deg
};
P[2249]{
   GP1:
	UF : 0, UT : 6,		CONFIG : 'N U T, 0, 0, 0',
	X =  426.001  mm,	Y =   -477.442  mm,	Z =   -229.167  mm,
	W =  90.000 deg,	P =   0.000 deg,	R =   90.000 deg
};
P[2250]{
   GP1:
	UF : 0, UT : 6,		CONFIG : 'N U T, 0, 0, 0',
	X =  426.951  mm,	Y =   -476.958  mm,	Z =   -229.008  mm,
	W =  90.000 deg,	P =   0.000 deg,	R =   90.000 deg
};
P[2251]{
   GP1:
	UF : 0, UT : 6,		CONFIG : 'N U T, 0, 0, 0',
	X =  428.184  mm,	Y =   -476.281  mm,	Z =   -228.923  mm,
	W =  90.000 deg,	P =   0.000 deg,	R =   90.000 deg
};
P[2252]{
   GP1:
	UF : 0, UT : 6,		CONFIG : 'N U T, 0, 0, 0',
	X =  429.239  mm,	Y =   -475.485  mm,	Z =   -229.377  mm,
	W =  90.000 deg,	P =   0.000 deg,	R =   90.000 deg
};
P[2253]{
   GP1:
	UF : 0, UT : 6,		CONFIG : 'N U T, 0, 0, 0',
	X =  430.726  mm,	Y =   -474.749  mm,	Z =   -229.080  mm,
	W =  90.000 deg,	P =   0.000 deg,	R =   90.000 deg
};
P[2254]{
   GP1:
	UF : 0, UT : 6,		CONFIG : 'N U T, 0, 0, 0',
	X =  431.781  mm,	Y =   -474.117  mm,	Z =   -229.137  mm,
	W =  90.000 deg,	P =   0.000 deg,	R =   90.000 deg
};
P[2255]{
   GP1:
	UF : 0, UT : 6,		CONFIG : 'N U T, 0, 0, 0',
	X =  432.802  mm,	Y =   -473.421  mm,	Z =   -229.392  mm,
	W =  90.000 deg,	P =   0.000 deg,	R =   90.000 deg
};
P[2256]{
   GP1:
	UF : 0, UT : 6,		CONFIG : 'N U T, 0, 0, 0',
	X =  435.250  mm,	Y =   -472.086  mm,	Z =   -229.205  mm,
	W =  90.000 deg,	P =   0.000 deg,	R =   90.000 deg
};
P[2257]{
   GP1:
	UF : 0, UT : 6,		CONFIG : 'N U T, 0, 0, 0',
	X =  437.802  mm,	Y =   -470.662  mm,	Z =   -229.083  mm,
	W =  90.000 deg,	P =   0.000 deg,	R =   90.000 deg
};
P[2258]{
   GP1:
	UF : 0, UT : 6,		CONFIG : 'N U T, 0, 0, 0',
	X =  439.158  mm,	Y =   -469.792  mm,	Z =   -229.295  mm,
	W =  90.000 deg,	P =   0.000 deg,	R =   90.000 deg
};
P[2259]{
   GP1:
	UF : 0, UT : 6,		CONFIG : 'N U T, 0, 0, 0',
	X =  441.656  mm,	Y =   -468.451  mm,	Z =   -229.051  mm,
	W =  90.000 deg,	P =   0.000 deg,	R =   90.000 deg
};
P[2260]{
   GP1:
	UF : 0, UT : 6,		CONFIG : 'N U T, 0, 0, 0',
	X =  443.229  mm,	Y =   -467.454  mm,	Z =   -229.266  mm,
	W =  90.000 deg,	P =   0.000 deg,	R =   90.000 deg
};
P[2261]{
   GP1:
	UF : 0, UT : 6,		CONFIG : 'N U T, 0, 0, 0',
	X =  444.845  mm,	Y =   -466.501  mm,	Z =   -229.314  mm,
	W =  90.000 deg,	P =   0.000 deg,	R =   90.000 deg
};
P[2262]{
   GP1:
	UF : 0, UT : 6,		CONFIG : 'N U T, 0, 0, 0',
	X =  447.932  mm,	Y =   -464.869  mm,	Z =   -228.946  mm,
	W =  90.000 deg,	P =   0.000 deg,	R =   90.000 deg
};
P[2263]{
   GP1:
	UF : 0, UT : 6,		CONFIG : 'N U T, 0, 0, 0',
	X =  450.483  mm,	Y =   -463.283  mm,	Z =   -229.220  mm,
	W =  90.000 deg,	P =   0.000 deg,	R =   90.000 deg
};
P[2264]{
   GP1:
	UF : 0, UT : 6,		CONFIG : 'N U T, 0, 0, 0',
	X =  452.017  mm,	Y =   -462.356  mm,	Z =   -229.320  mm,
	W =  90.000 deg,	P =   0.000 deg,	R =   90.000 deg
};
P[2265]{
   GP1:
	UF : 0, UT : 6,		CONFIG : 'N U T, 0, 0, 0',
	X =  452.675  mm,	Y =   -461.976  mm,	Z =   -229.323  mm,
	W =  90.000 deg,	P =   0.000 deg,	R =   90.000 deg
};
P[2266]{
   GP1:
	UF : 0, UT : 6,		CONFIG : 'N U T, 0, 0, 0',
	X =  455.201  mm,	Y =   -460.687  mm,	Z =   -228.910  mm,
	W =  90.000 deg,	P =   0.000 deg,	R =   90.000 deg
};
P[2267]{
   GP1:
	UF : 0, UT : 6,		CONFIG : 'N U T, 0, 0, 0',
	X =  456.568  mm,	Y =   -459.752  mm,	Z =   -229.264  mm,
	W =  90.000 deg,	P =   0.000 deg,	R =   90.000 deg
};
P[2268]{
   GP1:
	UF : 0, UT : 6,		CONFIG : 'N U T, 0, 0, 0',
	X =  458.044  mm,	Y =   -458.925  mm,	Z =   -229.204  mm,
	W =  90.000 deg,	P =   0.000 deg,	R =   90.000 deg
};
P[2269]{
   GP1:
	UF : 0, UT : 6,		CONFIG : 'N U T, 0, 0, 0',
	X =  459.334  mm,	Y =   -458.190  mm,	Z =   -229.180  mm,
	W =  90.000 deg,	P =   0.000 deg,	R =   90.000 deg
};
P[2270]{
   GP1:
	UF : 0, UT : 6,		CONFIG : 'N U T, 0, 0, 0',
	X =  460.129  mm,	Y =   -457.666  mm,	Z =   -229.336  mm,
	W =  90.000 deg,	P =   0.000 deg,	R =   90.000 deg
};
P[2271]{
   GP1:
	UF : 0, UT : 6,		CONFIG : 'N U T, 0, 0, 0',
	X =  461.684  mm,	Y =   -456.781  mm,	Z =   -229.305  mm,
	W =  90.000 deg,	P =   0.000 deg,	R =   90.000 deg
};
P[2272]{
   GP1:
	UF : 0, UT : 6,		CONFIG : 'N U T, 0, 0, 0',
	X =  462.817  mm,	Y =   -456.294  mm,	Z =   -228.901  mm,
	W =  90.000 deg,	P =   0.000 deg,	R =   90.000 deg
};
P[2273]{
   GP1:
	UF : 0, UT : 6,		CONFIG : 'N U T, 0, 0, 0',
	X =  464.685  mm,	Y =   -455.136  mm,	Z =   -229.092  mm,
	W =  90.000 deg,	P =   0.000 deg,	R =   90.000 deg
};
P[2274]{
   GP1:
	UF : 0, UT : 6,		CONFIG : 'N U T, 0, 0, 0',
	X =  465.379  mm,	Y =   -454.741  mm,	Z =   -229.080  mm,
	W =  90.000 deg,	P =   0.000 deg,	R =   90.000 deg
};
P[2275]{
   GP1:
	UF : 0, UT : 6,		CONFIG : 'N U T, 0, 0, 0',
	X =  468.747  mm,	Y =   -452.813  mm,	Z =   -229.039  mm,
	W =  90.000 deg,	P =   0.000 deg,	R =   90.000 deg
};
P[2276]{
   GP1:
	UF : 0, UT : 6,		CONFIG : 'N U T, 0, 0, 0',
	X =  469.967  mm,	Y =   -451.984  mm,	Z =   -229.341  mm,
	W =  90.000 deg,	P =   0.000 deg,	R =   90.000 deg
};
P[2277]{
   GP1:
	UF : 0, UT : 6,		CONFIG : 'N U T, 0, 0, 0',
	X =  470.687  mm,	Y =   -451.655  mm,	Z =   -229.131  mm,
	W =  90.000 deg,	P =   0.000 deg,	R =   90.000 deg
};
P[2278]{
   GP1:
	UF : 0, UT : 6,		CONFIG : 'N U T, 0, 0, 0',
	X =  471.996  mm,	Y =   -450.874  mm,	Z =   -229.193  mm,
	W =  90.000 deg,	P =   0.000 deg,	R =   90.000 deg
};
P[2279]{
   GP1:
	UF : 0, UT : 6,		CONFIG : 'N U T, 0, 0, 0',
	X =  472.567  mm,	Y =   -450.568  mm,	Z =   -229.134  mm,
	W =  90.000 deg,	P =   0.000 deg,	R =   90.000 deg
};
P[2280]{
   GP1:
	UF : 0, UT : 6,		CONFIG : 'N U T, 0, 0, 0',
	X =  473.790  mm,	Y =   -449.805  mm,	Z =   -229.273  mm,
	W =  90.000 deg,	P =   0.000 deg,	R =   90.000 deg
};
P[2281]{
   GP1:
	UF : 0, UT : 6,		CONFIG : 'N U T, 0, 0, 0',
	X =  475.060  mm,	Y =   -449.176  mm,	Z =   -229.018  mm,
	W =  90.000 deg,	P =   0.000 deg,	R =   90.000 deg
};
P[2282]{
   GP1:
	UF : 0, UT : 6,		CONFIG : 'N U T, 0, 0, 0',
	X =  476.620  mm,	Y =   -448.255  mm,	Z =   -229.068  mm,
	W =  90.000 deg,	P =   0.000 deg,	R =   90.000 deg
};
P[2283]{
   GP1:
	UF : 0, UT : 6,		CONFIG : 'N U T, 0, 0, 0',
	X =  477.104  mm,	Y =   -447.841  mm,	Z =   -229.397  mm,
	W =  90.000 deg,	P =   0.000 deg,	R =   90.000 deg
};
P[2284]{
   GP1:
	UF : 0, UT : 6,		CONFIG : 'N U T, 0, 0, 0',
	X =  479.135  mm,	Y =   -446.839  mm,	Z =   -228.979  mm,
	W =  90.000 deg,	P =   0.000 deg,	R =   90.000 deg
};
P[2285]{
   GP1:
	UF : 0, UT : 6,		CONFIG : 'N U T, 0, 0, 0',
	X =  479.869  mm,	Y =   -446.396  mm,	Z =   -229.029  mm,
	W =  90.000 deg,	P =   0.000 deg,	R =   90.000 deg
};
P[2286]{
   GP1:
	UF : 0, UT : 6,		CONFIG : 'N U T, 0, 0, 0',
